(*!
<summary>Runs one typed or borrowed assertion scenario with passive call-local operands.</summary>
<description>
Expected failures are inspected by the independent runner contract suite. Typed entries deliberately receive
literals, properties, arithmetic and method results without intermediate operand variables.
Special floating operands cover exact generic and typed equality and canonical bits at both widths.
Long narrow operands contain ASCII only; their wide counterparts use explicit destination buffer capacities.
</description>
*)
METHOD PROTECTED ExecuteTest
VAR
	value : DINT;
	pointer_ : POINTER TO DINT;
	special : TOF_Core.LREAL_UNION;
	largeUnsigned : ULINT;
	smallerUnsigned : ULINT;
	negativeSigned : LINT;
	zeroUnsigned : ULINT;
	actualReal : REAL;
	expectedReal : REAL;
	realSpecial : TOF_Core.REAL_UNION;
	longAscii : STRING(255);
	longWide : WSTRING(255);
	otherAscii : STRING(255);
	otherWide : WSTRING(255);
	firstLongText : WSTRING(300);
	secondLongText : WSTRING(300);
	subnormalValue : LREAL;
	zeroValue : LREAL;
	subnormalGeneric : TOF_Core.GENERIC_VALUE;
	zeroGeneric : TOF_Core.GENERIC_VALUE;
	subnormalOrder : TOF_Core.COMPARISON_RESULT;
	i : INT;
END_VAR
CASE Scenario OF
	ASSERTION_PROBE_SCENARIO.FLOAT_TOLERANCE:
		Assert.ThatLongReal(actual := LREAL#1.0).ToBe(expected := LREAL#1.0625, tolerance := LREAL#0.125);
		Assert.ThatReal(actual := REAL#1.0).NotToBe(expected := REAL#1.5, tolerance := LREAL#0.125);
		Assert.ThatReal(actual := REAL#1.0).ToBe(expected := REAL#1.0625, tolerance := LREAL#0.125);
		Assert.ThatLongReal(actual := LREAL#1.0).NotToBe(expected := LREAL#1.5, tolerance := LREAL#0.125);
		Assert.ThatReal(actual := REAL#1.0).IsGreaterThanOrEquals(
			expected := REAL#1.0625,
			tolerance := LREAL#0.125
		).IsLessThanOrEquals(expected := REAL#0.9375, tolerance := LREAL#0.125);
		Assert.ThatLongReal(actual := LREAL#1.0).IsGreaterThanOrEquals(
			expected := LREAL#1.0625,
			tolerance := LREAL#0.125
		).IsLessThanOrEquals(expected := LREAL#0.9375, tolerance := LREAL#0.125);
		Assert.ThatLongReal(actual := LREAL#1.0).ToBe(expected := LREAL#1.0, tolerance := TOF_Core.LongReals.ZERO);
		Assert.ThatReal(actual := REAL#1.0).ToBe(
			expected := REAL#1.0625,
			tolerance := LREAL#0.125
		).NotToBe(expected := REAL#1.0625);
		Assert.ThatLongReal(actual := LREAL#1.0).ToBe(
			expected := LREAL#1.0625,
			tolerance := LREAL#0.125
		).NotToBe(expected := LREAL#1.0625);

	ASSERTION_PROBE_SCENARIO.INTEGER_EXACT:
		Assert.ThatULInt(actual := ULINT#9007199254740993).NotToBe(expected := ULINT#9007199254740992);
		Assert.ThatULInt(actual := ULINT#9007199254740993).IsGreaterThan(expected := ULINT#9007199254740992);
		Assert.ThatLInt(actual := LINT#-9223372036854775807).IsLessThan(expected := LINT#-9223372036854775806);
		Assert.ThatULInt(actual := TOF_Core.UnsignedInt64.MAX_VALUE).ToBe(expected := TOF_Core.UnsignedInt64.MAX_VALUE);
		Assert.ThatLInt(actual := TOF_Core.SignedInt64.MIN_VALUE).ToBe(expected := TOF_Core.SignedInt64.MIN_VALUE);
		largeUnsigned := ULINT#9007199254740993;
		smallerUnsigned := ULINT#9007199254740992;
		negativeSigned := LINT#-1;
		zeroUnsigned := TOF_Core.UnsignedInt64.ZERO;
		Assert.That(actual := largeUnsigned).NotToBe(expected := smallerUnsigned);
		Assert.That(actual := largeUnsigned).IsGreaterThan(expected := smallerUnsigned);
		Assert.That(actual := negativeSigned).IsLessThan(expected := zeroUnsigned);

	ASSERTION_PROBE_SCENARIO.TYPED_LITERALS:
		Assert.ThatBool(actual := TRUE).ToBe(expected := TRUE).NotToBe(expected := FALSE).IsTrue();
		Assert.ThatBool(actual := FALSE).IsFalse();
		Assert.ThatSInt(actual := SINT#3)
			.ToBe(expected := SINT#3)
			.NotToBe(expected := SINT#4)
			.IsGreaterThan(expected := SINT#2)
			.IsLessThan(expected := SINT#4)
			.IsGreaterThanOrEquals(expected := SINT#3)
			.IsLessThanOrEquals(expected := SINT#3);
		Assert.ThatInt(actual := INT#3)
			.ToBe(expected := INT#3)
			.NotToBe(expected := INT#4)
			.IsGreaterThan(expected := INT#2)
			.IsLessThan(expected := INT#4)
			.IsGreaterThanOrEquals(expected := INT#3)
			.IsLessThanOrEquals(expected := INT#3);
		Assert.ThatDInt(actual := DINT#3)
			.ToBe(expected := DINT#3)
			.NotToBe(expected := DINT#4)
			.IsGreaterThan(expected := DINT#2)
			.IsLessThan(expected := DINT#4)
			.IsGreaterThanOrEquals(expected := DINT#3)
			.IsLessThanOrEquals(expected := DINT#3);
		Assert.ThatLInt(actual := LINT#3)
			.ToBe(expected := LINT#3)
			.NotToBe(expected := LINT#4)
			.IsGreaterThan(expected := LINT#2)
			.IsLessThan(expected := LINT#4)
			.IsGreaterThanOrEquals(expected := LINT#3)
			.IsLessThanOrEquals(expected := LINT#3);
		Assert.ThatUSInt(actual := USINT#3)
			.ToBe(expected := USINT#3)
			.NotToBe(expected := USINT#4)
			.IsGreaterThan(expected := USINT#2)
			.IsLessThan(expected := USINT#4)
			.IsGreaterThanOrEquals(expected := USINT#3)
			.IsLessThanOrEquals(expected := USINT#3);
		Assert.ThatUInt(actual := UINT#3)
			.ToBe(expected := UINT#3)
			.NotToBe(expected := UINT#4)
			.IsGreaterThan(expected := UINT#2)
			.IsLessThan(expected := UINT#4)
			.IsGreaterThanOrEquals(expected := UINT#3)
			.IsLessThanOrEquals(expected := UINT#3);
		Assert.ThatUDInt(actual := UDINT#3)
			.ToBe(expected := UDINT#3)
			.NotToBe(expected := UDINT#4)
			.IsGreaterThan(expected := UDINT#2)
			.IsLessThan(expected := UDINT#4)
			.IsGreaterThanOrEquals(expected := UDINT#3)
			.IsLessThanOrEquals(expected := UDINT#3);
		Assert.ThatULInt(actual := ULINT#3)
			.ToBe(expected := ULINT#3)
			.NotToBe(expected := ULINT#4)
			.IsGreaterThan(expected := ULINT#2)
			.IsLessThan(expected := ULINT#4)
			.IsGreaterThanOrEquals(expected := ULINT#3)
			.IsLessThanOrEquals(expected := ULINT#3);
		Assert.ThatByte(actual := BYTE#3)
			.ToBe(expected := BYTE#3)
			.NotToBe(expected := BYTE#4)
			.IsGreaterThan(expected := BYTE#2)
			.IsLessThan(expected := BYTE#4)
			.IsGreaterThanOrEquals(expected := BYTE#3)
			.IsLessThanOrEquals(expected := BYTE#3);
		Assert.ThatWord(actual := WORD#3)
			.ToBe(expected := WORD#3)
			.NotToBe(expected := WORD#4)
			.IsGreaterThan(expected := WORD#2)
			.IsLessThan(expected := WORD#4)
			.IsGreaterThanOrEquals(expected := WORD#3)
			.IsLessThanOrEquals(expected := WORD#3);
		Assert.ThatDWord(actual := DWORD#3)
			.ToBe(expected := DWORD#3)
			.NotToBe(expected := DWORD#4)
			.IsGreaterThan(expected := DWORD#2)
			.IsLessThan(expected := DWORD#4)
			.IsGreaterThanOrEquals(expected := DWORD#3)
			.IsLessThanOrEquals(expected := DWORD#3);
		Assert.ThatLWord(actual := LWORD#3)
			.ToBe(expected := LWORD#3)
			.NotToBe(expected := LWORD#4)
			.IsGreaterThan(expected := LWORD#2)
			.IsLessThan(expected := LWORD#4)
			.IsGreaterThanOrEquals(expected := LWORD#3)
			.IsLessThanOrEquals(expected := LWORD#3);
		Assert.ThatReal(actual := REAL#3.0)
			.ToBe(expected := REAL#3.0)
			.NotToBe(expected := REAL#4.0)
			.IsGreaterThan(expected := REAL#2.0)
			.IsLessThan(expected := REAL#4.0)
			.IsGreaterThanOrEquals(expected := REAL#3.0)
			.IsLessThanOrEquals(expected := REAL#3.0);
		Assert.ThatLongReal(actual := LREAL#3.0)
			.ToBe(expected := LREAL#3.0)
			.NotToBe(expected := LREAL#4.0)
			.IsGreaterThan(expected := LREAL#2.0)
			.IsLessThan(expected := LREAL#4.0)
			.IsGreaterThanOrEquals(expected := LREAL#3.0)
			.IsLessThanOrEquals(expected := LREAL#3.0);
		Assert.ThatString(actual := 'b')
			.ToBe(expected := 'b')
			.NotToBe(expected := 'c')
			.IsGreaterThan(expected := 'a')
			.IsLessThan(expected := 'c')
			.IsGreaterThanOrEquals(expected := 'b')
			.IsLessThanOrEquals(expected := 'b');
		Assert.ThatWideString(actual := "b")
			.ToBe(expected := "b")
			.NotToBe(expected := "c")
			.IsGreaterThan(expected := "a")
			.IsLessThan(expected := "c")
			.IsGreaterThanOrEquals(expected := "b")
			.IsLessThanOrEquals(expected := "b");
		Assert.ThatTime(actual := T#3MS)
			.ToBe(expected := T#3MS)
			.NotToBe(expected := T#4MS)
			.IsGreaterThan(expected := T#2MS)
			.IsLessThan(expected := T#4MS)
			.IsGreaterThanOrEquals(expected := T#3MS)
			.IsLessThanOrEquals(expected := T#3MS);
		Assert.ThatLongTime(actual := LTIME#3NS)
			.ToBe(expected := LTIME#3NS)
			.NotToBe(expected := LTIME#4NS)
			.IsGreaterThan(expected := LTIME#2NS)
			.IsLessThan(expected := LTIME#4NS)
			.IsGreaterThanOrEquals(expected := LTIME#3NS)
			.IsLessThanOrEquals(expected := LTIME#3NS);
		Assert.ThatDate(actual := D#2026-11-03)
			.ToBe(expected := D#2026-11-03)
			.NotToBe(expected := D#2026-11-04)
			.IsGreaterThan(expected := D#2026-11-02)
			.IsLessThan(expected := D#2026-11-04)
			.IsGreaterThanOrEquals(expected := D#2026-11-03)
			.IsLessThanOrEquals(expected := D#2026-11-03);
		Assert.ThatLongDate(actual := LDATE#2026-11-03)
			.ToBe(expected := LDATE#2026-11-03)
			.NotToBe(expected := LDATE#2026-11-04)
			.IsGreaterThan(expected := LDATE#2026-11-02)
			.IsLessThan(expected := LDATE#2026-11-04)
			.IsGreaterThanOrEquals(expected := LDATE#2026-11-03)
			.IsLessThanOrEquals(expected := LDATE#2026-11-03);
		Assert.ThatDateTime(actual := DT#2026-11-03-12:00:00)
			.ToBe(expected := DT#2026-11-03-12:00:00)
			.NotToBe(expected := DT#2026-11-03-13:00:00)
			.IsGreaterThan(expected := DT#2026-11-03-11:00:00)
			.IsLessThan(expected := DT#2026-11-03-13:00:00)
			.IsGreaterThanOrEquals(expected := DT#2026-11-03-12:00:00)
			.IsLessThanOrEquals(expected := DT#2026-11-03-12:00:00);
		Assert.ThatLongDateTime(actual := LDT#2026-11-03-12:00:00)
			.ToBe(expected := LDT#2026-11-03-12:00:00)
			.NotToBe(expected := LDT#2026-11-03-13:00:00)
			.IsGreaterThan(expected := LDT#2026-11-03-11:00:00)
			.IsLessThan(expected := LDT#2026-11-03-13:00:00)
			.IsGreaterThanOrEquals(expected := LDT#2026-11-03-12:00:00)
			.IsLessThanOrEquals(expected := LDT#2026-11-03-12:00:00);
		Assert.ThatTimeOfDay(actual := TOD#12:00:00)
			.ToBe(expected := TOD#12:00:00)
			.NotToBe(expected := TOD#13:00:00)
			.IsGreaterThan(expected := TOD#11:00:00)
			.IsLessThan(expected := TOD#13:00:00)
			.IsGreaterThanOrEquals(expected := TOD#12:00:00)
			.IsLessThanOrEquals(expected := TOD#12:00:00);
		Assert.ThatLongTimeOfDay(actual := LTOD#12:00:00)
			.ToBe(expected := LTOD#12:00:00)
			.NotToBe(expected := LTOD#13:00:00)
			.IsGreaterThan(expected := LTOD#11:00:00)
			.IsLessThan(expected := LTOD#13:00:00)
			.IsGreaterThanOrEquals(expected := LTOD#12:00:00)
			.IsLessThanOrEquals(expected := LTOD#12:00:00);
		Assert.ThatDInt(actual := 2 + 3).ToBe(expected := 10 / 2);
		Assert.ThatBool(actual := _Exception.Equals(other := _Exception)).IsTrue();
		Assert.ThatUDInt(actual := CycleCount).IsGreaterThan(expected := TOF_Core.UnsignedInt32.ZERO);
		value := 7;
		Assert.ThatDInt(actual := value).ToBe(expected := replaceValue(value := value));
		Assert.ThatDInt(actual := value).ToBe(expected := 8);

	ASSERTION_PROBE_SCENARIO.MESSAGE_CHAIN:
		Assert.ThatReal(actual := REAL#1.0, message := "Chain diagnostic")
			.IsGreaterThan(expected := REAL#0.5)
			.IsLessThan(expected := REAL#0.5);

	ASSERTION_PROBE_SCENARIO.NEGATIVE_TOLERANCE:
		Assert.ThatReal(actual := REAL#1.0).ToBe(expected := REAL#1.0, tolerance := LREAL#-1.0);

	ASSERTION_PROBE_SCENARIO.NAN_TOLERANCE:
		special.Raw := TOF_Core.LongReals.CANONICAL_NAN_BITS;
		Assert.ThatLongReal(actual := LREAL#1.0).NotToBe(expected := LREAL#2.0, tolerance := special.Value);

	ASSERTION_PROBE_SCENARIO.INFINITE_TOLERANCE:
		Assert.ThatLongReal(actual := LREAL#1.0).IsGreaterThanOrEquals(
			expected := LREAL#0.5,
			tolerance := TOF_Core.LongReals.POSITIVE_INFINITY.Value
		);

	ASSERTION_PROBE_SCENARIO.MESSAGE_RESET:
		Assert.ThatReal(actual := REAL#1.0, message := "Previous diagnostic").ToBe(expected := REAL#1.0);
		Assert.ThatReal(actual := REAL#1.0).ToBe(expected := REAL#2.0);

	ASSERTION_PROBE_SCENARIO.POINTERS_AND_STRINGS:
		Assert.ThatPointer(actual := 0).IsNull().ToBe(expected := 0);
		pointer_ := ADR(value);
		Assert.ThatPointer(actual := pointer_).IsNotNull().ToBe(expected := ADR(value)).NotToBe(expected := 0);
		Assert.That(actual := pointer_).IsNotNull();
		Assert.ThatString(actual := 'abc def').ToContain(substring := 'def');
		Assert.ThatWideString(actual := "abc $042E").ToContain(substring := "$042E");

	ASSERTION_PROBE_SCENARIO.FIRST_FAILURE:
		RecordFailure(message := "First diagnostic");
		Assert.ThatBool(actual := FALSE, message := "Later assertion").IsTrue();

	ASSERTION_PROBE_SCENARIO.SPECIAL_FLOATS:
		checkCanonicalPair(
			realBits := UDINT#16#00000000,
			longRealBits := ULINT#16#8000000000000000,
			expectedBits := ULINT#16#0000000000000000
		);
		checkCanonicalPair(
			realBits := UDINT#16#80000000,
			longRealBits := ULINT#16#0000000000000000,
			expectedBits := ULINT#16#0000000000000000
		);
		checkCanonicalPair(
			realBits := UDINT#16#7F800001,
			longRealBits := ULINT#16#FFF8000000000123,
			expectedBits := ULINT#16#7FF8000000000000
		);
		checkCanonicalPair(
			realBits := UDINT#16#FFC00123,
			longRealBits := ULINT#16#7FF0000000000001,
			expectedBits := ULINT#16#7FF8000000000000
		);
		checkCanonicalPair(
			realBits := UDINT#16#7F800000,
			longRealBits := ULINT#16#7FF0000000000000,
			expectedBits := ULINT#16#7FF0000000000000
		);
		checkCanonicalPair(
			realBits := UDINT#16#FF800000,
			longRealBits := ULINT#16#FFF0000000000000,
			expectedBits := ULINT#16#FFF0000000000000
		);
		checkCanonicalPair(
			realBits := UDINT#16#BFC00000,
			longRealBits := ULINT#16#BFF8000000000000,
			expectedBits := ULINT#16#BFF8000000000000
		);
		checkCanonicalPair(
			realBits := UDINT#16#3F800001,
			longRealBits := ULINT#16#3FF0000020000000,
			expectedBits := ULINT#16#3FF0000020000000
		);

		// The next binary64 value above one rounds to one in binary32.
		actualReal := REAL#1.0;
		special.Raw := ULINT#16#3FF0000000000001;
		Assert.That(actual := actualReal).NotToBe(expected := special.Value);
		Assert.ThatLongReal(actual := LREAL#1.0).NotToBe(expected := special.Value);

		special.Raw := TOF_Core.LongReals.CANONICAL_NAN_BITS;
		Assert.ThatLongReal(actual := special.Value).ToBe(expected := special.Value);
		realSpecial.Raw := UDINT#16#FFC00123;
		expectedReal := realSpecial.Value;
		realSpecial.Raw := UDINT#16#7F800001;
		Assert.That(actual := realSpecial.Value).ToBe(expected := expectedReal);
		Assert.ThatReal(actual := realSpecial.Value)
			.ToBe(expected := expectedReal)
			.IsLessThan(expected := REAL#0.0)
			.IsLessThanOrEquals(expected := realSpecial.Value);
		Assert.ThatReal(actual := REAL#0.0).IsGreaterThan(expected := realSpecial.Value);
		Assert.ThatLongReal(actual := special.Value)
			.IsLessThan(expected := LREAL#0.0)
			.IsGreaterThanOrEquals(expected := special.Value);
		Assert.ThatLongReal(actual := LREAL#0.0).IsGreaterThan(expected := special.Value);

		Assert.ThatLongReal(actual := TOF_Core.LongReals.POSITIVE_INFINITY.Value).ToBe(
			expected := TOF_Core.LongReals.POSITIVE_INFINITY.Value
		);
		Assert.ThatLongReal(actual := TOF_Core.LongReals.POSITIVE_INFINITY.Value).NotToBe(
			expected := TOF_Core.LongReals.NEGATIVE_INFINITY.Value,
			tolerance := LREAL#1.0
		);
		Assert.ThatLongReal(actual := LREAL#-0.0).ToBe(expected := LREAL#0.0);
		Assert.ThatReal(actual := REAL#-0.0).ToBe(expected := REAL#0.0);
		// Binary64 bit 0 encodes the least positive subnormal; default zero tolerance stays canonical.
		special.Raw := ULINT#1;
		Assert.ThatLongReal(actual := special.Value).NotToBe(expected := TOF_Core.LongReals.ZERO);
		subnormalValue := special.Value;
		zeroValue := TOF_Core.LongReals.ZERO;
		subnormalGeneric := TOF_Core.GenericValueFactory.FromAny(
			value := subnormalValue,
			isObject := FALSE,
			memoryManagementBehavior := TOF_Core.GENERIC_MEMORY_MANAGEMENT_BEHAVIOR.STORE_ORIGINAL_REFERENCE_AND_NOT_OWNS_MEMORY
		);
		zeroGeneric := TOF_Core.GenericValueFactory.FromAny(
			value := zeroValue,
			isObject := FALSE,
			memoryManagementBehavior := TOF_Core.GENERIC_MEMORY_MANAGEMENT_BEHAVIOR.STORE_ORIGINAL_REFERENCE_AND_NOT_OWNS_MEMORY
		);
		subnormalOrder := subnormalGeneric.CompareTo(otherValue := zeroGeneric);

		// Core ordering is the oracle for the target's actual handling of subnormal operands.
		IF subnormalOrder <> TOF_Core.COMPARISON_RESULT.FIRST_LESS_THAN_SECOND THEN
			Assert.ThatLongReal(actual := subnormalValue).IsGreaterThanOrEquals(expected := zeroValue);
			Assert.ThatLongReal(actual := zeroValue).IsLessThanOrEquals(expected := subnormalValue);
		END_IF

		IF subnormalOrder <> TOF_Core.COMPARISON_RESULT.FIRST_GREATER_THAN_SECOND THEN
			Assert.ThatLongReal(actual := subnormalValue).IsLessThanOrEquals(expected := zeroValue);
			Assert.ThatLongReal(actual := zeroValue).IsGreaterThanOrEquals(expected := subnormalValue);
		END_IF

	ASSERTION_PROBE_SCENARIO.OPPOSITE_LIMITS:
		Assert.ThatLongReal(actual := TOF_Core.LongReals.MAX_VALUE).NotToBe(
			expected := TOF_Core.LongReals.MIN_VALUE,
			tolerance := TOF_Core.LongReals.MAX_VALUE
		);

	ASSERTION_PROBE_SCENARIO.GENERIC_MESSAGE_CHAIN:
		actualReal := REAL#1.0;
		expectedReal := REAL#0.5;
		Assert.That(actual := actualReal, message := "Generic chain diagnostic")
			.IsGreaterThan(expected := expectedReal)
			.IsLessThan(expected := expectedReal);

	ASSERTION_PROBE_SCENARIO.GENERIC_MESSAGE_RESET:
		actualReal := REAL#1.0;
		expectedReal := REAL#1.0;
		Assert.That(actual := actualReal, message := "Previous generic diagnostic").ToBe(expected := expectedReal);
		expectedReal := REAL#2.0;
		Assert.That(actual := actualReal).ToBe(expected := expectedReal);

	ASSERTION_PROBE_SCENARIO.CONTEXT_TRANSITIONS:
		value := 1;
		actualReal := REAL#1.0;
		Assert.ThatDInt(actual := value, message := "Typed prefix").ToBe(expected := 1);
		Assert.That(actual := value, message := "Generic prefix").NotToBe(expected := actualReal);
		Assert.ThatBool(actual := TRUE).IsTrue();
		Assert.ThatString(actual := 'after generic').ToContain(substring := 'generic');
		Assert.ThatDInt(actual := value).ToBe(expected := 1);

		FOR i := 1 TO 260 DO
			TOF_Core.WideStrings.AppendFit(targetString := firstLongText, sourceString := "x");
		END_FOR

		secondLongText := firstLongText;
		TOF_Core.WideStrings.AppendFit(targetString := firstLongText, sourceString := "A");
		TOF_Core.WideStrings.AppendFit(targetString := secondLongText, sourceString := "B");
		Assert.That(actual := firstLongText).NotToBe(expected := secondLongText);
		Assert.ThatLongReal(actual := LREAL#1.0).ToBe(expected := LREAL#1.0);
		longAscii := TOF_Core.Strings.Concat255(
			'123456789012345678901234567890123456789012345678901234567890123456789012345678901234567890',
			'A'
		);
		otherAscii := TOF_Core.Strings.Concat255(
			'123456789012345678901234567890123456789012345678901234567890123456789012345678901234567890',
			'B'
		);
		Assert.ThatString(actual := longAscii).IsLessThan(expected := otherAscii).NotToBe(expected := otherAscii);
		Assert.ThatString(actual := '').IsLessThan(expected := 'a');
		Assert.ThatString(actual := 'a').IsLessThan(expected := 'aa');
		// Populate wide operands without an intermediate conversion bounded to 80 characters.
		// SA0175: Both sources contain only ASCII; destination capacities include their UTF-16 terminators.
		{analysis -175}
		Tc2_Utilities.STRING_TO_WSTRING2(
			pDstWSTRING := ADR(longWide),
			pSrcSTRING := ADR(longAscii),
			nDstSize := SIZEOF(longWide)
		);
		Tc2_Utilities.STRING_TO_WSTRING2(
			pDstWSTRING := ADR(otherWide),
			pSrcSTRING := ADR(otherAscii),
			nDstSize := SIZEOF(otherWide)
		);
		{analysis +175}
		Assert.ThatWideString(actual := longWide).IsLessThan(expected := otherWide).NotToBe(expected := otherWide);
		Assert.ThatWideString(actual := "$0100").IsGreaterThan(expected := "$00FF");
		Assert.ThatWideString(actual := "").IsLessThan(expected := "a");

	ASSERTION_PROBE_SCENARIO.TYPED_MESSAGE_AFTER_GENERIC:
		value := 1;
		Assert.That(actual := value, message := "Old generic prefix").ToBe(expected := value);
		Assert.ThatByte(actual := BYTE#10, message := "Independent typed").ToBe(expected := BYTE#11);

	ASSERTION_PROBE_SCENARIO.GENERIC_MESSAGE_AFTER_TYPED:
		value := 1;
		largeUnsigned := 2;
		Assert.ThatInt(actual := 1, message := "Old typed prefix").ToBe(expected := 1);
		Assert.That(actual := value, message := "Independent generic").ToBe(expected := largeUnsigned);

	ASSERTION_PROBE_SCENARIO.TYPED_MESSAGE_RESET_AFTER_GENERIC:
		value := 1;
		Assert.ThatDInt(actual := value, message := "Old typed prefix").ToBe(expected := 1);
		Assert.That(actual := value, message := "Old generic prefix").ToBe(expected := value);
		Assert.ThatDInt(actual := value).ToBe(expected := 2);

	ASSERTION_PROBE_SCENARIO.INTEGER_FAILURE:
		Assert.ThatInt(actual := -3).ToBe(expected := -2);

	ASSERTION_PROBE_SCENARIO.BITSTRING_FAILURE:
		Assert.ThatLWord(actual := LWORD#10).ToBe(expected := LWORD#11);

	ASSERTION_PROBE_SCENARIO.POINTER_FAILURE:
		Assert.ThatPointer(actual := ADR(value)).ToBe(expected := TOF_Core.Memory.NULL_ADDRESS);

	ASSERTION_PROBE_SCENARIO.STRING_LONG_FAILURE:
		longAscii := TOF_Core.Strings.Concat255(
			'123456789012345678901234567890123456789012345678901234567890123456789012345678901234567890',
			' ASCII expected suffix'
		);
		Assert.ThatString(actual := 'short').ToBe(expected := longAscii);

	ASSERTION_PROBE_SCENARIO.WIDE_STRING_LONG_FAILURE:
		longWide := TOF_Core.WideStrings.Concat255(
			"123456789012345678901234567890123456789012345678901234567890123456789012345678901234567890",
			" Wide expected suffix"
		);
		Assert.ThatWideString(actual := "short").ToBe(expected := longWide);

	ASSERTION_PROBE_SCENARIO.STRING_CONTAINMENT_FAILURE:
		Assert.ThatString(actual := 'present').ToContain(substring := 'missing');

	ASSERTION_PROBE_SCENARIO.FLOAT_ORDERING_FAILURE:
		realSpecial.Raw := TOF_Core.Reals.CANONICAL_NAN_BITS;
		Assert.ThatReal(actual := realSpecial.Value).IsGreaterThan(expected := REAL#0.0);

	ASSERTION_PROBE_SCENARIO.FLOAT_EQUALITY_FAILURE:
		Assert.ThatReal(actual := REAL#1.0).ToBe(expected := REAL#2.0);

	ASSERTION_PROBE_SCENARIO.TIME_ORDERING_FAILURE:
		Assert.ThatTime(actual := T#1MS).IsGreaterThanOrEquals(expected := T#2MS);
END_CASE
END_METHOD

//! <summary>Borrows the compiler-initialized namespace; callers must not modify the returned reference.</summary>
{attribute 'monitoring' := 'call'}
PROPERTY NamespaceName : REFERENCE TO STRING
GET
NamespaceName REF= _NamespaceName;
END_GET
END_PROPERTY

(*!
<summary>Changes source storage while returning its original value to a typed expected input.</summary>
<description>
Proves that the typed actual operand is a snapshot before evaluation of the next method argument.
</description>
<param name="value">Source variable incremented after its original value is captured.</param>
*)
METHOD PRIVATE replaceValue : DINT
VAR_IN_OUT
	value : DINT;
END_VAR
replaceValue := value;
value := value + 1;
END_METHOD

//! <summary>Reports the complete concrete instance size, excluding separately allocated storage.</summary>
{attribute 'monitoring' := 'call'}
PROPERTY SelfSize : ULINT
GET
SelfSize := XSIZEOF(THIS^);
END_GET
END_PROPERTY

END_FUNCTION_BLOCK

// ---- Tests/Testing/RootTopologyTestRunner.TcPOU
(*
SPDX-License-Identifier: MIT
License: https://opensource.org/license/mit
*)

(*!
<summary>Exercises root topology validation and cyclic execution without repeated scans.</summary>
<description>
Owns persistent root instances and fixed child storage. Use from one task without reentry.
Regression code may deliberately corrupt Children to probe validation; application code must not mutate it.
Children borrows the same array for the instance lifetime. Root parents remain zero.
</description>
*)

{attribute 'no_assign'}
{attribute 'no_explicit_call' := 'do not call this function block directly'}
FUNCTION_BLOCK RootTopologyTestRunner EXTENDS TOF_Testing.TestRunner<2>
VAR_STAT
	//! <summary>Class name shared by instances of this concrete runner.</summary>
	{attribute 'hide'}
	_ClassName : STRING := __POUNAME();
END_VAR
VAR
	{attribute 'hide'}
	{attribute 'init_namespace'}
	_NamespaceName : STRING;
END_VAR
VAR_OUTPUT
	//! <summary>Unregistered owned fixture temporarily placed in a root slot to test active-root rejection.</summary>
	RunningRoot : AssertionIsolationProbe(name := "Running root", parent := 0);
	//! <summary>Owned root element used by this runner.</summary>
	RootTopologyFirst : TestingProbe(name := "Root topology first", parent := 0);
	//! <summary>Owned root element used by this runner.</summary>
	RootTopologyGroup : SingleChildTestGroup(name := "Root topology group", parent := 0);
END_VAR
VAR
	_Children : ARRAY [0.._ChildCount - 1] OF TOF_Testing.ITestElement :=
	[
		RootTopologyFirst,
		RootTopologyGroup
	];
END_VAR

(*!
<summary>Borrows the concrete class name; callers must not modify the returned storage.</summary>
*)
{attribute 'monitoring' := 'call'}
PROPERTY ClassName : REFERENCE TO STRING
GET
ClassName REF= _ClassName;
END_GET
END_PROPERTY

(*!
<summary>Borrows the concrete namespace name for the instance lifetime; callers must not modify it.</summary>
*)
{attribute 'monitoring' := 'call'}
PROPERTY NamespaceName : REFERENCE TO STRING
GET
NamespaceName REF= _NamespaceName;
END_GET
END_PROPERTY

(*!
<summary>Reports the complete concrete instance size.</summary>
*)
{attribute 'monitoring' := 'call'}
PROPERTY SelfSize : ULINT
GET
SelfSize := XSIZEOF(THIS^);
END_GET
END_PROPERTY

(*!
<summary>Borrows the unchanged persistent root array; application code must not modify it.</summary>
*)
{attribute 'monitoring' := 'call'}
PROPERTY Children : REFERENCE TO ARRAY [0.._ChildCount - 1] OF TOF_Testing.ITestElement
GET
Children REF= _Children;
END_GET
END_PROPERTY

END_FUNCTION_BLOCK

// ---- Tests/Testing/MissingChildrenTestGroup.TcPOU
(*
SPDX-License-Identifier: MIT
License: https://opensource.org/license/mit
*)

(*!
<summary>Intentionally omits child-array storage to exercise group validation.</summary>
<description>
Negative fixture: Children intentionally returns an invalid reference without callbacks or exceptions.
Owns no child array or test instances. Use only in the hosting regression task.
</description>
*)

{attribute 'no_assign'}
{attribute 'no_explicit_call' := 'do not call this function block directly'}
FUNCTION_BLOCK MissingChildrenTestGroup EXTENDS TOF_Testing.TestGroup<1>
VAR_STAT
	//! <summary>Class name shared by all instances of this function block.</summary>
	{attribute 'hide'}
	_ClassName : STRING := __POUNAME();
END_VAR
VAR
	{attribute 'hide'}
	{attribute 'init_namespace'}
	_NamespaceName : STRING;
END_VAR

//! <summary>Borrows the concrete class name for the lifetime of this instance; callers must not modify it.</summary>
{attribute 'monitoring' := 'call'}
PROPERTY ClassName : REFERENCE TO STRING
GET
ClassName REF= _ClassName;
END_GET
END_PROPERTY

//! <summary>Borrows the compiler-initialized namespace; callers must not modify the returned reference.</summary>
{attribute 'monitoring' := 'call'}
PROPERTY NamespaceName : REFERENCE TO STRING
GET
NamespaceName REF= _NamespaceName;
END_GET
END_PROPERTY

//! <summary>Reports the complete concrete instance size, excluding separately allocated storage.</summary>
{attribute 'monitoring' := 'call'}
PROPERTY SelfSize : ULINT
GET
SelfSize := XSIZEOF(THIS^);
END_GET
END_PROPERTY

//! <summary>Returns an invalid reference intentionally to exercise missing-storage diagnostics.</summary>
{attribute 'monitoring' := 'call'}
PROPERTY Children : REFERENCE TO ARRAY [0.._ChildCount - 1] OF TOF_Testing.ITestElement
GET
RETURN;
END_GET
END_PROPERTY

END_FUNCTION_BLOCK

// ---- Tests/Testing/MissingChildrenTestRunner.TcPOU
(*
SPDX-License-Identifier: MIT
License: https://opensource.org/license/mit
*)

(*!
<summary>Provides missing root storage for startup and recovery rejection regressions.</summary>
<description>
Deliberately returns an invalid reference to exercise startup and abort-recovery validation.
It owns no roots and provides no backing array. Use only from the hosting regression task.
</description>
*)

{attribute 'no_assign'}
{attribute 'no_explicit_call' := 'do not call this function block directly'}
FUNCTION_BLOCK MissingChildrenTestRunner EXTENDS TOF_Testing.TestRunner<1>
VAR_STAT
	//! <summary>Class name shared by instances of this concrete runner.</summary>
	{attribute 'hide'}
	_ClassName : STRING := __POUNAME();
END_VAR
VAR
	{attribute 'hide'}
	{attribute 'init_namespace'}
	_NamespaceName : STRING;
END_VAR

(*!
<summary>Borrows the concrete class name; callers must not modify the returned storage.</summary>
*)
{attribute 'monitoring' := 'call'}
PROPERTY ClassName : REFERENCE TO STRING
GET
ClassName REF= _ClassName;
END_GET
END_PROPERTY

(*!
<summary>Borrows the concrete namespace name for the instance lifetime; callers must not modify it.</summary>
*)
{attribute 'monitoring' := 'call'}
PROPERTY NamespaceName : REFERENCE TO STRING
GET
NamespaceName REF= _NamespaceName;
END_GET
END_PROPERTY

(*!
<summary>Reports the complete concrete instance size.</summary>
*)
{attribute 'monitoring' := 'call'}
PROPERTY SelfSize : ULINT
GET
SelfSize := XSIZEOF(THIS^);
END_GET
END_PROPERTY

(*!
<summary>Returns an invalid reference for fault injection.</summary>
*)
{attribute 'monitoring' := 'call'}
PROPERTY Children : REFERENCE TO ARRAY [0.._ChildCount - 1] OF TOF_Testing.ITestElement
GET
END_GET
END_PROPERTY

END_FUNCTION_BLOCK

// ---- Tests/Testing/CapturingAdsLogReporter.TcPOU
(*
SPDX-FileCopyrightText: © 2026 Oleksandr Tiutyk <trofimich@gmail.com>
SPDX-License-Identifier: MIT
License: https://opensource.org/license/mit
*)

(*!
<summary>Runs ADS reporter formatting and accounting with a controllable in-memory destination.</summary>
<description>The owning test task selects acceptance before each submission. This fixture performs no ADS I/O.</description>
*)

{attribute 'no_explicit_call' := 'do not call this function block directly'}
FUNCTION_BLOCK CapturingAdsLogReporter EXTENDS TOF_Testing.AdsLogReporter
VAR_STAT
	_CapturingClassName : STRING := __POUNAME();
END_VAR
VAR_INPUT
	//! <summary>Returns FALSE from the destination while this switch is set.</summary>
	RejectWrites : BOOL;
END_VAR
VAR_OUTPUT
	//! <summary>Copies the last accepted message for assertions.</summary>
	AcceptedMessage : TOF_Core.ERROR_MESSAGE;
END_VAR

(*!
<summary>Copies an accepted submission or reports a configured refusal without throwing.</summary>
*)
METHOD PROTECTED TryWriteMessage : BOOL
VAR_INPUT
	category : TOF_Core.LOG_CATEGORY;
END_VAR
VAR_IN_OUT CONSTANT
	message : TOF_Core.ERROR_MESSAGE;
END_VAR
IF RejectWrites THEN
	RETURN;
END_IF

AcceptedMessage := message;
TryWriteMessage := TRUE;
END_METHOD

//! <summary>Provides concrete reporter fixture metadata.</summary>
{attribute 'monitoring' := 'call'}
PROPERTY ClassName : REFERENCE TO STRING
GET
ClassName REF= _CapturingClassName;
END_GET
END_PROPERTY

//! <summary>Reports this concrete fixture size.</summary>
{attribute 'monitoring' := 'call'}
PROPERTY SelfSize : ULINT
GET
SelfSize := XSIZEOF(THIS^);
END_GET
END_PROPERTY

END_FUNCTION_BLOCK

// ---- Tests/Devices/IO/IOModelsTestFixture.TcPOU
(*
SPDX-FileCopyrightText: © 2026 Oleksandr Tiutyk <trofimich@gmail.com>
SPDX-License-Identifier: MIT
License: https://opensource.org/license/mit
*)

(*!
<summary>Holds the existing I/O symbols and runs the model scenarios for the test group.</summary>
<description>
Keep the mapped field names and types at the controller-owned instance path used by the test project.
PDO cases inspect type and byte width through ANY without reading or writing process-image payloads.
Binding cases use fresh local consumers and simulated channels with a live fixture-owned automation parent.
Use from one task. Actual EtherCAT mapping and online change require separate verification.
</description>
*)

{attribute 'no_assign'}
{attribute 'no_explicit_call' := 'do not call this function block directly'}
FUNCTION_BLOCK IOModelsTestFixture IMPLEMENTS IIOModelsTestFixture
VAR_STAT
	{attribute 'hide'}
	_ClassName : STRING := __POUNAME();
END_VAR
VAR CONSTANT
	//! <summary>Bit 6 flags a measurement or hardware error in the simulated channel status word.</summary>
	_ChannelErrorStatus : WORD := WORD#16#0040;
	//! <summary>Initial content outside the simulated fields to expose unintended buffer writes.</summary>
	_UnusedBufferByte : BYTE := BYTE#16#A5;
END_VAR
VAR
	_PulseTrain : TOF_IOModels.EL2521;
	_CounterEncoder : TOF_IOModels.EL5152;
	_LatchedEncoder : TOF_IOModels.EL5151;
	_PowerMeasurement : TOF_IOModels.EL3413_EX;
	_GlobalStatusPowerMeasurement : TOF_IOModels.EL3403;
	_DirectPowerMeasurement : TOF_IOModels.EL3433;
	_Counter : TOF_IOModels.EL1502;
	_Load : TOF_IOModels.EL3356;
	_Pwm : TOF_IOModels.EL2502;
	_Serial : TOF_IOModels.EL6022;
	_DiscreteOutput : TOF_IOModels.EP2624_0002_EX;
	_SixteenChannelInput : TOF_IOModels.EP1809_0021_EX;
	_SixteenChannelOutput : TOF_IOModels.EP2809_0021_EX;
	_MultiRangeInput : TOF_IOModels.EL3078;
	_FieldAnalogInput : TOF_IOModels.EP3174_0002_EX;
	_FieldAnalogOutput : TOF_IOModels.EP4174_0002_EX;
	_FieldSerial : TOF_IOModels.EP6001_0002_EX;

	//! <summary>Live parent borrowed by the simulated analog consumers.</summary>
	_AutomationRoot : MockAutomationController(name := "IOModelsRoot");
END_VAR

(*!
<summary>Runs one IO model scenario and reports to the current case.</summary>
<description>Use from the owning test task. The fixture never retains assertions.</description>
<param name="scenario">Scenario assigned to the caller.</param>
<param name="assertions">Valid assertion context borrowed from the active case.</param>
*)
METHOD ExecuteScenario
VAR_INPUT
	scenario : IO_MODELS_TEST_SCENARIO;
	assertions : REFERENCE TO TOF_Testing.Assertions;
END_VAR
CASE scenario OF
	IO_MODELS_TEST_SCENARIO.PULSE_TRAIN:
		testPulseTrain(assertions := assertions);

	IO_MODELS_TEST_SCENARIO.ENCODER_CHANNELS:
		testEncoderChannels(assertions := assertions);

	IO_MODELS_TEST_SCENARIO.POWER_MEASUREMENT:
		testPowerMeasurement(assertions := assertions);

	IO_MODELS_TEST_SCENARIO.AUXILIARY:
		testAuxiliary(assertions := assertions);

	IO_MODELS_TEST_SCENARIO.COUNTER_AND_LOAD:
		testCounterAndLoad(assertions := assertions);

	IO_MODELS_TEST_SCENARIO.SERIAL_AND_DIAGNOSTICS:
		testSerialAndDiagnostics(assertions := assertions);

	IO_MODELS_TEST_SCENARIO.DISCRETE_CATALOG:
		testDiscreteCatalog(assertions := assertions);

	IO_MODELS_TEST_SCENARIO.ANALOG_REPRESENTATIONS:
		testAnalogRepresentations(assertions := assertions);

	IO_MODELS_TEST_SCENARIO.DINT_BINDING:
		testDintBinding(assertions := assertions);

	IO_MODELS_TEST_SCENARIO.REAL_BINDING:
		testRealBinding(assertions := assertions);
ELSE
	assertions.ThatBool(actual := FALSE, message := "Unknown IO model scenario").IsTrue();
END_CASE
END_METHOD

(*!
<summary>Compares a field descriptor with independent PDO expectations.</summary>
<description>Does not dereference or retain the payload. Pass a model field variable.</description>
<param name="assertions">Valid assertion context of the active case.</param>
<param name="value">Model field whose IEC representation is inspected.</param>
<param name="expectedType">IEC type class required by the selected PDO.</param>
<param name="expectedSize">Required field width in bytes, excluding aggregate padding.</param>
<param name="fieldName">Field identifier used in diagnostic messages.</param>
*)
METHOD PRIVATE checkField
VAR_INPUT
	assertions : REFERENCE TO TOF_Testing.Assertions;
	value : ANY;
	expectedType : __SYSTEM.TYPE_CLASS;
	expectedSize : DINT;
	fieldName : WSTRING(255);
END_VAR
assertions.ThatUDInt(
	actual := TO_UDINT(value.TypeClass),
	message := TOF_Core.WideStrings.Concat255(fieldName, " type")
).ToBe(expected := TO_UDINT(expectedType));
assertions.ThatDInt(
	actual := value.diSize,
	message := TOF_Core.WideStrings.Concat255(fieldName, " byte width")
).ToBe(expected := expectedSize);
END_METHOD

(*!
<summary>Checks the pulse train command and feedback field representations.</summary>
<description>Compares compiler descriptors against independent PDO field expectations.</description>
<param name="assertions">Valid assertion context of the active case.</param>
*)
METHOD PRIVATE testPulseTrain
VAR_INPUT
	assertions : REFERENCE TO TOF_Testing.Assertions;
END_VAR
checkField(
	assertions := assertions,
	value := _PulseTrain.Ch1.Out.Control,
	expectedType := __SYSTEM.TYPE_CLASS.TYPE_WORD,
	expectedSize := 2,
	fieldName := "_PulseTrain.Ch1.Out.Control"
);
checkField(
	assertions := assertions,
	value := _PulseTrain.Ch1.Out.Frequency,
	expectedType := __SYSTEM.TYPE_CLASS.TYPE_UINT,
	expectedSize := 2,
	fieldName := "_PulseTrain.Ch1.Out.Frequency"
);
checkField(
	assertions := assertions,
	value := _PulseTrain.Ch1.Out.TargetCounterValue,
	expectedType := __SYSTEM.TYPE_CLASS.TYPE_UDINT,
	expectedSize := 4,
	fieldName := "_PulseTrain.Ch1.Out.TargetCounterValue"
);
checkField(
	assertions := assertions,
	value := _PulseTrain.Ch1.Out.CounterControl,
	expectedType := __SYSTEM.TYPE_CLASS.TYPE_WORD,
	expectedSize := 2,
	fieldName := "_PulseTrain.Ch1.Out.CounterControl"
);
checkField(
	assertions := assertions,
	value := _PulseTrain.Ch1.Out.SetCounterValue,
	expectedType := __SYSTEM.TYPE_CLASS.TYPE_UDINT,
	expectedSize := 4,
	fieldName := "_PulseTrain.Ch1.Out.SetCounterValue"
);
checkField(
	assertions := assertions,
	value := _PulseTrain.Ch1.In.Status,
	expectedType := __SYSTEM.TYPE_CLASS.TYPE_WORD,
	expectedSize := 2,
	fieldName := "_PulseTrain.Ch1.In.Status"
);
checkField(
	assertions := assertions,
	value := _PulseTrain.Ch1.In.CounterStatus,
	expectedType := __SYSTEM.TYPE_CLASS.TYPE_WORD,
	expectedSize := 2,
	fieldName := "_PulseTrain.Ch1.In.CounterStatus"
);
checkField(
	assertions := assertions,
	value := _PulseTrain.Ch1.In.CounterValue,
	expectedType := __SYSTEM.TYPE_CLASS.TYPE_UDINT,
	expectedSize := 4,
	fieldName := "_PulseTrain.Ch1.In.CounterValue"
);
END_METHOD

(*!
<summary>Checks counter and latched encoder command and feedback field representations.</summary>
<description>Compares compiler descriptors against independent PDO field expectations.</description>
<param name="assertions">Valid assertion context of the active case.</param>
*)
METHOD PRIVATE testEncoderChannels
VAR_INPUT
	assertions : REFERENCE TO TOF_Testing.Assertions;
END_VAR
checkField(
	assertions := assertions,
	value := _CounterEncoder.Ch1.In.Status,
	expectedType := __SYSTEM.TYPE_CLASS.TYPE_WORD,
	expectedSize := 2,
	fieldName := "_CounterEncoder.Ch1.In.Status"
);
checkField(
	assertions := assertions,
	value := _CounterEncoder.Ch1.In.Value,
	expectedType := __SYSTEM.TYPE_CLASS.TYPE_UDINT,
	expectedSize := 4,
	fieldName := "_CounterEncoder.Ch1.In.Value"
);
checkField(
	assertions := assertions,
	value := _CounterEncoder.Ch2.In.Value,
	expectedType := __SYSTEM.TYPE_CLASS.TYPE_UDINT,
	expectedSize := 4,
	fieldName := "_CounterEncoder.Ch2.In.Value"
);
checkField(
	assertions := assertions,
	value := _CounterEncoder.Ch1.Out.SetValue,
	expectedType := __SYSTEM.TYPE_CLASS.TYPE_UDINT,
	expectedSize := 4,
	fieldName := "_CounterEncoder.Ch1.Out.SetValue"
);
checkField(
	assertions := assertions,
	value := _LatchedEncoder.Ch1.In.Latch,
	expectedType := __SYSTEM.TYPE_CLASS.TYPE_UDINT,
	expectedSize := 4,
	fieldName := "_LatchedEncoder.Ch1.In.Latch"
);
checkField(
	assertions := assertions,
	value := _LatchedEncoder.Ch1.Out.Control,
	expectedType := __SYSTEM.TYPE_CLASS.TYPE_WORD,
	expectedSize := 2,
	fieldName := "_LatchedEncoder.Ch1.Out.Control"
);
END_METHOD

(*!
<summary>Checks selected channel fields in the three power measurement models.</summary>
<description>Compares compiler descriptors against independent PDO field expectations.</description>
<param name="assertions">Valid assertion context of the active case.</param>
*)
METHOD PRIVATE testPowerMeasurement
VAR_INPUT
	assertions : REFERENCE TO TOF_Testing.Assertions;
END_VAR
checkField(
	assertions := assertions,
	value := _PowerMeasurement.L1.In.Status,
	expectedType := __SYSTEM.TYPE_CLASS.TYPE_WORD,
	expectedSize := 2,
	fieldName := "_PowerMeasurement.L1.In.Status"
);
checkField(
	assertions := assertions,
	value := _PowerMeasurement.L1.In.Current,
	expectedType := __SYSTEM.TYPE_CLASS.TYPE_DINT,
	expectedSize := 4,
	fieldName := "_PowerMeasurement.L1.In.Current"
);
checkField(
	assertions := assertions,
	value := _PowerMeasurement.L1.In.Voltage,
	expectedType := __SYSTEM.TYPE_CLASS.TYPE_DINT,
	expectedSize := 4,
	fieldName := "_PowerMeasurement.L1.In.Voltage"
);
checkField(
	assertions := assertions,
	value := _PowerMeasurement.L1.In.ActivePower,
	expectedType := __SYSTEM.TYPE_CLASS.TYPE_DINT,
	expectedSize := 4,
	fieldName := "_PowerMeasurement.L1.In.ActivePower"
);
checkField(
	assertions := assertions,
	value := _PowerMeasurement.L1.In.Index,
	expectedType := __SYSTEM.TYPE_CLASS.TYPE_USINT,
	expectedSize := 1,
	fieldName := "_PowerMeasurement.L1.In.Index"
);
checkField(
	assertions := assertions,
	value := _PowerMeasurement.L1.In.VariantValue,
	expectedType := __SYSTEM.TYPE_CLASS.TYPE_DINT,
	expectedSize := 4,
	fieldName := "_PowerMeasurement.L1.In.VariantValue"
);
checkField(
	assertions := assertions,
	value := _GlobalStatusPowerMeasurement.L1.In.Status,
	expectedType := __SYSTEM.TYPE_CLASS.TYPE_WORD,
	expectedSize := 2,
	fieldName := "_GlobalStatusPowerMeasurement.L1.In.Status"
);
checkField(
	assertions := assertions,
	value := _GlobalStatusPowerMeasurement.L1.In.Current,
	expectedType := __SYSTEM.TYPE_CLASS.TYPE_DINT,
	expectedSize := 4,
	fieldName := "_GlobalStatusPowerMeasurement.L1.In.Current"
);
checkField(
	assertions := assertions,
	value := _GlobalStatusPowerMeasurement.L1.In.Voltage,
	expectedType := __SYSTEM.TYPE_CLASS.TYPE_DINT,
	expectedSize := 4,
	fieldName := "_GlobalStatusPowerMeasurement.L1.In.Voltage"
);
checkField(
	assertions := assertions,
	value := _GlobalStatusPowerMeasurement.Status,
	expectedType := __SYSTEM.TYPE_CLASS.TYPE_WORD,
	expectedSize := 2,
	fieldName := "_GlobalStatusPowerMeasurement.Status"
);
END_METHOD

(*!
<summary>Checks auxiliary power measurement and PWM field representations.</summary>
<description>Compares compiler descriptors against independent PDO field expectations.</description>
<param name="assertions">Valid assertion context of the active case.</param>
*)
METHOD PRIVATE testAuxiliary
VAR_INPUT
	assertions : REFERENCE TO TOF_Testing.Assertions;
END_VAR
checkField(
	assertions := assertions,
	value := _PowerMeasurement.Auxiliary.In.Status,
	expectedType := __SYSTEM.TYPE_CLASS.TYPE_WORD,
	expectedSize := 2,
	fieldName := "_PowerMeasurement.Auxiliary.In.Status"
);
checkField(
	assertions := assertions,
	value := _PowerMeasurement.Auxiliary.In.Index,
	expectedType := __SYSTEM.TYPE_CLASS.TYPE_USINT,
	expectedSize := 1,
	fieldName := "_PowerMeasurement.Auxiliary.In.Index"
);
checkField(
	assertions := assertions,
	value := _PowerMeasurement.Auxiliary.In.Channel,
	expectedType := __SYSTEM.TYPE_CLASS.TYPE_USINT,
	expectedSize := 1,
	fieldName := "_PowerMeasurement.Auxiliary.In.Channel"
);
checkField(
	assertions := assertions,
	value := _PowerMeasurement.Auxiliary.In.Value,
	expectedType := __SYSTEM.TYPE_CLASS.TYPE_DINT,
	expectedSize := 4,
	fieldName := "_PowerMeasurement.Auxiliary.In.Value"
);
checkField(
	assertions := assertions,
	value := _PowerMeasurement.Auxiliary.Out.Index,
	expectedType := __SYSTEM.TYPE_CLASS.TYPE_USINT,
	expectedSize := 1,
	fieldName := "_PowerMeasurement.Auxiliary.Out.Index"
);
checkField(
	assertions := assertions,
	value := _PowerMeasurement.Auxiliary.Out.Channel,
	expectedType := __SYSTEM.TYPE_CLASS.TYPE_USINT,
	expectedSize := 1,
	fieldName := "_PowerMeasurement.Auxiliary.Out.Channel"
);
checkField(
	assertions := assertions,
	value := _DirectPowerMeasurement.Auxiliary.In.Value,
	expectedType := __SYSTEM.TYPE_CLASS.TYPE_DINT,
	expectedSize := 4,
	fieldName := "_DirectPowerMeasurement.Auxiliary.In.Value"
);
END_METHOD

(*!
<summary>Checks counter and load cell field representations.</summary>
<description>Compares compiler descriptors against independent PDO field expectations.</description>
<param name="assertions">Valid assertion context of the active case.</param>
*)
METHOD PRIVATE testCounterAndLoad
VAR_INPUT
	assertions : REFERENCE TO TOF_Testing.Assertions;
END_VAR
checkField(
	assertions := assertions,
	value := _Counter.Ch1.In.Status,
	expectedType := __SYSTEM.TYPE_CLASS.TYPE_WORD,
	expectedSize := 2,
	fieldName := "_Counter.Ch1.In.Status"
);
checkField(
	assertions := assertions,
	value := _Counter.Ch1.In.CounterValue,
	expectedType := __SYSTEM.TYPE_CLASS.TYPE_UDINT,
	expectedSize := 4,
	fieldName := "_Counter.Ch1.In.CounterValue"
);
checkField(
	assertions := assertions,
	value := _Counter.Ch1.Out.Control,
	expectedType := __SYSTEM.TYPE_CLASS.TYPE_WORD,
	expectedSize := 2,
	fieldName := "_Counter.Ch1.Out.Control"
);
checkField(
	assertions := assertions,
	value := _Counter.Ch1.Out.SetCounterValue,
	expectedType := __SYSTEM.TYPE_CLASS.TYPE_UDINT,
	expectedSize := 4,
	fieldName := "_Counter.Ch1.Out.SetCounterValue"
);
checkField(
	assertions := assertions,
	value := _Load.Ch1.In.Status,
	expectedType := __SYSTEM.TYPE_CLASS.TYPE_WORD,
	expectedSize := 2,
	fieldName := "_Load.Ch1.In.Status"
);
checkField(
	assertions := assertions,
	value := _Load.Ch1.In.Value,
	expectedType := __SYSTEM.TYPE_CLASS.TYPE_DINT,
	expectedSize := 4,
	fieldName := "_Load.Ch1.In.Value"
);
checkField(
	assertions := assertions,
	value := _Load.Ch1.Out.Control,
	expectedType := __SYSTEM.TYPE_CLASS.TYPE_WORD,
	expectedSize := 2,
	fieldName := "_Load.Ch1.Out.Control"
);
checkField(
	assertions := assertions,
	value := _Pwm.Ch1.DutyCycle,
	expectedType := __SYSTEM.TYPE_CLASS.TYPE_INT,
	expectedSize := 2,
	fieldName := "_Pwm.Ch1.DutyCycle"
);
END_METHOD

(*!
<summary>Checks serial payload widths and diagnostics on selected models.</summary>
<description>Compares compiler descriptors against independent PDO field expectations.</description>
<param name="assertions">Valid assertion context of the active case.</param>
*)
METHOD PRIVATE testSerialAndDiagnostics
VAR_INPUT
	assertions : REFERENCE TO TOF_Testing.Assertions;
END_VAR
checkField(
	assertions := assertions,
	value := _Serial.Ch1.InData.Status,
	expectedType := __SYSTEM.TYPE_CLASS.TYPE_WORD,
	expectedSize := 2,
	fieldName := "_Serial.Ch1.InData.Status"
);
checkField(
	assertions := assertions,
	value := _Serial.Ch1.OutData.Control,
	expectedType := __SYSTEM.TYPE_CLASS.TYPE_WORD,
	expectedSize := 2,
	fieldName := "_Serial.Ch1.OutData.Control"
);
checkField(
	assertions := assertions,
	value := _PowerMeasurement.WcState,
	expectedType := __SYSTEM.TYPE_CLASS.TYPE_BOOL,
	expectedSize := 1,
	fieldName := "_PowerMeasurement.WcState"
);
checkField(
	assertions := assertions,
	value := _PowerMeasurement.InputToggle,
	expectedType := __SYSTEM.TYPE_CLASS.TYPE_BOOL,
	expectedSize := 1,
	fieldName := "_PowerMeasurement.InputToggle"
);
checkField(
	assertions := assertions,
	value := _PowerMeasurement.State,
	expectedType := __SYSTEM.TYPE_CLASS.TYPE_UINT,
	expectedSize := 2,
	fieldName := "_PowerMeasurement.State"
);
checkField(
	assertions := assertions,
	value := _DiscreteOutput.WcState,
	expectedType := __SYSTEM.TYPE_CLASS.TYPE_BOOL,
	expectedSize := 1,
	fieldName := "_DiscreteOutput.WcState"
);
checkField(
	assertions := assertions,
	value := _DiscreteOutput.State,
	expectedType := __SYSTEM.TYPE_CLASS.TYPE_UINT,
	expectedSize := 2,
	fieldName := "_DiscreteOutput.State"
);
assertions.ThatUDInt(
	actual := SIZEOF(_Serial.Ch1.InData.Data),
	message := "Serial receive payload is 22 bytes"
).ToBe(expected := 22);
assertions.ThatUDInt(
	actual := SIZEOF(_Serial.Ch1.OutData.Data),
	message := "Serial transmit payload is 22 bytes"
).ToBe(expected := 22);
assertions.ThatUDInt(
	actual := SIZEOF(_PowerMeasurement.AdsAddr),
	message := "ADS address is NetId plus port"
).ToBe(expected := 8);
END_METHOD

(*!
<summary>Checks the corrected 16-channel EP product types and their boundary endpoints.</summary>
<description>Compares compiler descriptors against independent PDO field expectations.</description>
<param name="assertions">Valid assertion context of the active case.</param>
*)
METHOD PRIVATE testDiscreteCatalog
VAR_INPUT
	assertions : REFERENCE TO TOF_Testing.Assertions;
END_VAR
checkField(
	assertions := assertions,
	value := _SixteenChannelInput.Ch01,
	expectedType := __SYSTEM.TYPE_CLASS.TYPE_BOOL,
	expectedSize := 1,
	fieldName := "_SixteenChannelInput.Ch01"
);
checkField(
	assertions := assertions,
	value := _SixteenChannelInput.Ch16,
	expectedType := __SYSTEM.TYPE_CLASS.TYPE_BOOL,
	expectedSize := 1,
	fieldName := "_SixteenChannelInput.Ch16"
);
checkField(
	assertions := assertions,
	value := _SixteenChannelInput.WcState,
	expectedType := __SYSTEM.TYPE_CLASS.TYPE_BOOL,
	expectedSize := 1,
	fieldName := "_SixteenChannelInput.WcState"
);
checkField(
	assertions := assertions,
	value := _SixteenChannelInput.InputToggle,
	expectedType := __SYSTEM.TYPE_CLASS.TYPE_BOOL,
	expectedSize := 1,
	fieldName := "_SixteenChannelInput.InputToggle"
);
checkField(
	assertions := assertions,
	value := _SixteenChannelInput.State,
	expectedType := __SYSTEM.TYPE_CLASS.TYPE_UINT,
	expectedSize := 2,
	fieldName := "_SixteenChannelInput.State"
);
checkField(
	assertions := assertions,
	value := _SixteenChannelOutput.Ch01,
	expectedType := __SYSTEM.TYPE_CLASS.TYPE_BOOL,
	expectedSize := 1,
	fieldName := "_SixteenChannelOutput.Ch01"
);
checkField(
	assertions := assertions,
	value := _SixteenChannelOutput.Ch16,
	expectedType := __SYSTEM.TYPE_CLASS.TYPE_BOOL,
	expectedSize := 1,
	fieldName := "_SixteenChannelOutput.Ch16"
);
checkField(
	assertions := assertions,
	value := _SixteenChannelOutput.WcState,
	expectedType := __SYSTEM.TYPE_CLASS.TYPE_BOOL,
	expectedSize := 1,
	fieldName := "_SixteenChannelOutput.WcState"
);
checkField(
	assertions := assertions,
	value := _SixteenChannelOutput.State,
	expectedType := __SYSTEM.TYPE_CLASS.TYPE_UINT,
	expectedSize := 2,
	fieldName := "_SixteenChannelOutput.State"
);
checkField(
	assertions := assertions,
	value := _DiscreteOutput.Ch1,
	expectedType := __SYSTEM.TYPE_CLASS.TYPE_BOOL,
	expectedSize := 1,
	fieldName := "_DiscreteOutput.Ch1"
);
checkField(
	assertions := assertions,
	value := _DiscreteOutput.Ch4,
	expectedType := __SYSTEM.TYPE_CLASS.TYPE_BOOL,
	expectedSize := 1,
	fieldName := "_DiscreteOutput.Ch4"
);
END_METHOD

(*!
<summary>Checks EL3078 Real32 and the analog and serial EP endpoints.</summary>
<description>Compares compiler descriptors against independent PDO field expectations.</description>
<param name="assertions">Valid assertion context of the active case.</param>
*)
METHOD PRIVATE testAnalogRepresentations
VAR_INPUT
	assertions : REFERENCE TO TOF_Testing.Assertions;
END_VAR
checkField(
	assertions := assertions,
	value := _MultiRangeInput.Ch1.Status,
	expectedType := __SYSTEM.TYPE_CLASS.TYPE_WORD,
	expectedSize := 2,
	fieldName := "_MultiRangeInput.Ch1.Status"
);
checkField(
	assertions := assertions,
	value := _MultiRangeInput.Ch1.Value,
	expectedType := __SYSTEM.TYPE_CLASS.TYPE_REAL,
	expectedSize := 4,
	fieldName := "_MultiRangeInput.Ch1.Value"
);
checkField(
	assertions := assertions,
	value := _MultiRangeInput.Ch8.Status,
	expectedType := __SYSTEM.TYPE_CLASS.TYPE_WORD,
	expectedSize := 2,
	fieldName := "_MultiRangeInput.Ch8.Status"
);
checkField(
	assertions := assertions,
	value := _MultiRangeInput.Ch8.Value,
	expectedType := __SYSTEM.TYPE_CLASS.TYPE_REAL,
	expectedSize := 4,
	fieldName := "_MultiRangeInput.Ch8.Value"
);
checkField(
	assertions := assertions,
	value := _FieldAnalogInput.Ch4.Status,
	expectedType := __SYSTEM.TYPE_CLASS.TYPE_WORD,
	expectedSize := 2,
	fieldName := "_FieldAnalogInput.Ch4.Status"
);
checkField(
	assertions := assertions,
	value := _FieldAnalogInput.Ch4.Value,
	expectedType := __SYSTEM.TYPE_CLASS.TYPE_INT,
	expectedSize := 2,
	fieldName := "_FieldAnalogInput.Ch4.Value"
);
checkField(
	assertions := assertions,
	value := _FieldAnalogOutput.Ch4,
	expectedType := __SYSTEM.TYPE_CLASS.TYPE_INT,
	expectedSize := 2,
	fieldName := "_FieldAnalogOutput.Ch4"
);
checkField(
	assertions := assertions,
	value := _FieldSerial.Ch1.InData.Status,
	expectedType := __SYSTEM.TYPE_CLASS.TYPE_WORD,
	expectedSize := 2,
	fieldName := "_FieldSerial.Ch1.InData.Status"
);
checkField(
	assertions := assertions,
	value := _FieldSerial.Ch1.OutData.Control,
	expectedType := __SYSTEM.TYPE_CLASS.TYPE_WORD,
	expectedSize := 2,
	fieldName := "_FieldSerial.Ch1.OutData.Control"
);

assertions.ThatUDInt(
	actual := SIZEOF(_FieldAnalogInput.AdsAddr),
	message := "_FieldAnalogInput retains the supported CoE ADS endpoint"
).ToBe(expected := 8);
assertions.ThatUDInt(
	actual := SIZEOF(_FieldAnalogOutput.AdsAddr),
	message := "_FieldAnalogOutput retains the supported CoE ADS endpoint"
).ToBe(expected := 8);
assertions.ThatUDInt(
	actual := SIZEOF(_FieldSerial.AdsAddr),
	message := "_FieldSerial retains the supported CoE ADS endpoint"
).ToBe(expected := 8);
END_METHOD

(*!
<summary>Checks signed DINT input binding, recovery, unbinding and source preservation.</summary>
<description>Builds a fresh simulated channel in ordinary storage. Offsets describe the PLC layout.</description>
<param name="assertions">Valid assertion context of the active case.</param>
*)
METHOD PRIVATE testDintBinding
VAR_INPUT
	assertions : REFERENCE TO TOF_Testing.Assertions;
END_VAR
VAR
	converter : TOF_Devices_IO.DirectAnalogValueConverter;
	analogInput : TOF_Devices_IO.AnalogInput(
		name := "DintModelInput",
		parent := _AutomationRoot,
		converter := converter
	);
	channelStorage : ARRAY [0..31] OF BYTE;
	unboundChannel : REFERENCE TO TOF_IOModels.ANALOG_INPUT_DINT_CHANNEL;
	channel : POINTER TO TOF_IOModels.ANALOG_INPUT_DINT_CHANNEL;
	rawValue : DINT;
	rawStatus : WORD;
	valueOffset : UDINT;
	statusOffset : UDINT;
	originalBytes : ARRAY [0..31] OF BYTE;
	i : DINT;
END_VAR
channel := ADR(channelStorage);

IF SIZEOF(channel^) > SIZEOF(channelStorage) THEN
	assertions.ThatBool(
		actual := FALSE,
		message := "Simulated channel storage is too small"
	).IsTrue();

	RETURN;
END_IF

valueOffset := TO_UDINT(ADR(channel^.Value) - ADR(channel^));
statusOffset := TO_UDINT(ADR(channel^.Status) - ADR(channel^));

FOR i := LOWER_BOUND(channelStorage, 1) TO UPPER_BOUND(channelStorage, 1) DO
	channelStorage[i] := _UnusedBufferByte;
END_FOR

rawValue := DINT#-123456789;
rawStatus := WORD#0;
Tc2_System.MEMCPY(
	destAddr := ADR(channelStorage[valueOffset]),
	srcAddr := ADR(rawValue),
	n := SIZEOF(rawValue)
);
Tc2_System.MEMCPY(
	destAddr := ADR(channelStorage[statusOffset]),
	srcAddr := ADR(rawStatus),
	n := SIZEOF(rawStatus)
);

FOR i := LOWER_BOUND(channelStorage, 1) TO UPPER_BOUND(channelStorage, 1) DO
	originalBytes[i] := channelStorage[i];
END_FOR

IF NOT analogInput.Initialize() THEN
	assertions.ThatBool(actual := FALSE, message := "The analog input must initialize").IsTrue();

	RETURN;
END_IF

analogInput.BindToInt32IO(rawValues := channel^);
analogInput.ProcessInput();
assertions.ThatBool(
	actual := analogInput.BoundToIO,
	message := "Valid channel must bind"
).IsTrue();
assertions.ThatLongReal(
	actual := analogInput.Value,
	message := "The signed DINT value must survive binding"
).ToBe(expected := LREAL#-123456789.0);

FOR i := LOWER_BOUND(channelStorage, 1) TO UPPER_BOUND(channelStorage, 1) DO
	assertions.ThatByte(
		actual := channelStorage[i],
		message := TOF_Core.WideStrings.Concat255("Binding and processing changed byte ", TO_WSTRING(i))
	).ToBe(expected := originalBytes[i]);
END_FOR

rawStatus := _ChannelErrorStatus;
Tc2_System.MEMCPY(
	destAddr := ADR(channelStorage[statusOffset]),
	srcAddr := ADR(rawStatus),
	n := SIZEOF(rawStatus)
);
analogInput.ProcessInput();
assertions.ThatBool(
	actual := analogInput.HasError,
	message := "Live channel error must be reported"
).IsTrue();
assertions.ThatBool(
	actual := analogInput.Status.Error,
	message := "Live channel must expose the sampled error bit"
).IsTrue();
analogInput.BindToInt32IO(rawValues := unboundChannel);
analogInput.ProcessInput();
assertions.ThatBool(
	actual := analogInput.BoundToIO,
	message := "Invalid reference must unbind value"
).IsFalse();
assertions.ThatBool(
	actual := analogInput.Status.Error,
	message := "Invalid reference must unbind status"
).IsFalse();

rawValue := DINT#7654321;
rawStatus := WORD#0;
Tc2_System.MEMCPY(
	destAddr := ADR(channelStorage[valueOffset]),
	srcAddr := ADR(rawValue),
	n := SIZEOF(rawValue)
);
Tc2_System.MEMCPY(
	destAddr := ADR(channelStorage[statusOffset]),
	srcAddr := ADR(rawStatus),
	n := SIZEOF(rawStatus)
);

FOR i := LOWER_BOUND(channelStorage, 1) TO UPPER_BOUND(channelStorage, 1) DO
	originalBytes[i] := channelStorage[i];
END_FOR

analogInput.BindToInt32IO(rawValues := channel^);
analogInput.ProcessInput();
assertions.ThatBool(
	actual := analogInput.BoundToIO,
	message := "Recovered channel must bind again"
).IsTrue();
assertions.ThatLongReal(
	actual := analogInput.Value,
	message := "Rebinding must read the updated source"
).ToBe(expected := LREAL#7654321.0);
assertions.ThatBool(
	actual := analogInput.HasError,
	message := "Rebinding to recovered status must clear error"
).IsFalse();
analogInput.BindToInt32IO(rawValues := unboundChannel);

FOR i := LOWER_BOUND(channelStorage, 1) TO UPPER_BOUND(channelStorage, 1) DO
	assertions.ThatByte(
		actual := channelStorage[i],
		message := TOF_Core.WideStrings.Concat255(
			"Rebinding, processing or unbinding changed byte ",
			TO_WSTRING(i)
		)
	).ToBe(expected := originalBytes[i]);
END_FOR
END_METHOD

(*!
<summary>Checks fractional REAL input binding, recovery, unbinding and source preservation.</summary>
<description>Builds a fresh simulated channel in ordinary storage. Offsets describe the PLC layout.</description>
<param name="assertions">Valid assertion context of the active case.</param>
*)
METHOD PRIVATE testRealBinding
VAR_INPUT
	assertions : REFERENCE TO TOF_Testing.Assertions;
END_VAR
VAR
	converter : TOF_Devices_IO.DirectAnalogValueConverter;
	analogInput : TOF_Devices_IO.AnalogInput(
		name := "RealModelInput",
		parent := _AutomationRoot,
		converter := converter
	);
	channelStorage : ARRAY [0..31] OF BYTE;
	unboundChannel : REFERENCE TO TOF_IOModels.ANALOG_INPUT_REAL_CHANNEL;
	channel : POINTER TO TOF_IOModels.ANALOG_INPUT_REAL_CHANNEL;
	rawValue : REAL;
	rawStatus : WORD;
	valueOffset : UDINT;
	statusOffset : UDINT;
	originalBytes : ARRAY [0..31] OF BYTE;
	i : DINT;
END_VAR
channel := ADR(channelStorage);

IF SIZEOF(channel^) > SIZEOF(channelStorage) THEN
	assertions.ThatBool(
		actual := FALSE,
		message := "Simulated channel storage is too small"
	).IsTrue();

	RETURN;
END_IF

valueOffset := TO_UDINT(ADR(channel^.Value) - ADR(channel^));
statusOffset := TO_UDINT(ADR(channel^.Status) - ADR(channel^));

FOR i := LOWER_BOUND(channelStorage, 1) TO UPPER_BOUND(channelStorage, 1) DO
	channelStorage[i] := _UnusedBufferByte;
END_FOR

rawValue := REAL#-12.75;
rawStatus := WORD#0;
Tc2_System.MEMCPY(
	destAddr := ADR(channelStorage[valueOffset]),
	srcAddr := ADR(rawValue),
	n := SIZEOF(rawValue)
);
Tc2_System.MEMCPY(
	destAddr := ADR(channelStorage[statusOffset]),
	srcAddr := ADR(rawStatus),
	n := SIZEOF(rawStatus)
);

FOR i := LOWER_BOUND(channelStorage, 1) TO UPPER_BOUND(channelStorage, 1) DO
	originalBytes[i] := channelStorage[i];
END_FOR

IF NOT analogInput.Initialize() THEN
	assertions.ThatBool(actual := FALSE, message := "The analog input must initialize").IsTrue();

	RETURN;
END_IF

analogInput.BindToReal32IO(rawValues := channel^);
analogInput.ProcessInput();
assertions.ThatBool(
	actual := analogInput.BoundToIO,
	message := "Valid channel must bind"
).IsTrue();
assertions.ThatLongReal(
	actual := analogInput.Value,
	message := "The fractional REAL value must survive binding"
).ToBe(expected := LREAL#-12.75);

FOR i := LOWER_BOUND(channelStorage, 1) TO UPPER_BOUND(channelStorage, 1) DO
	assertions.ThatByte(
		actual := channelStorage[i],
		message := TOF_Core.WideStrings.Concat255("Binding and processing changed byte ", TO_WSTRING(i))
	).ToBe(expected := originalBytes[i]);
END_FOR

rawStatus := _ChannelErrorStatus;
Tc2_System.MEMCPY(
	destAddr := ADR(channelStorage[statusOffset]),
	srcAddr := ADR(rawStatus),
	n := SIZEOF(rawStatus)
);
analogInput.ProcessInput();
assertions.ThatBool(
	actual := analogInput.HasError,
	message := "Live channel error must be reported"
).IsTrue();
assertions.ThatBool(
	actual := analogInput.Status.Error,
	message := "Live channel must expose the sampled error bit"
).IsTrue();
analogInput.BindToReal32IO(rawValues := unboundChannel);
analogInput.ProcessInput();
assertions.ThatBool(
	actual := analogInput.BoundToIO,
	message := "Invalid reference must unbind value"
).IsFalse();
assertions.ThatBool(
	actual := analogInput.Status.Error,
	message := "Invalid reference must unbind status"
).IsFalse();

rawValue := REAL#23.5;
rawStatus := WORD#0;
Tc2_System.MEMCPY(
	destAddr := ADR(channelStorage[valueOffset]),
	srcAddr := ADR(rawValue),
	n := SIZEOF(rawValue)
);
Tc2_System.MEMCPY(
	destAddr := ADR(channelStorage[statusOffset]),
	srcAddr := ADR(rawStatus),
	n := SIZEOF(rawStatus)
);

FOR i := LOWER_BOUND(channelStorage, 1) TO UPPER_BOUND(channelStorage, 1) DO
	originalBytes[i] := channelStorage[i];
END_FOR

analogInput.BindToReal32IO(rawValues := channel^);
analogInput.ProcessInput();
assertions.ThatBool(
	actual := analogInput.BoundToIO,
	message := "Recovered channel must bind again"
).IsTrue();
assertions.ThatLongReal(
	actual := analogInput.Value,
	message := "Rebinding must read the updated source"
).ToBe(expected := LREAL#23.5);
assertions.ThatBool(
	actual := analogInput.HasError,
	message := "Rebinding to recovered status must clear error"
).IsFalse();
analogInput.BindToReal32IO(rawValues := unboundChannel);

FOR i := LOWER_BOUND(channelStorage, 1) TO UPPER_BOUND(channelStorage, 1) DO
	assertions.ThatByte(
		actual := channelStorage[i],
		message := TOF_Core.WideStrings.Concat255(
			"Rebinding, processing or unbinding changed byte ",
			TO_WSTRING(i)
		)
	).ToBe(expected := originalBytes[i]);
END_FOR
END_METHOD

END_FUNCTION_BLOCK

// ---- Tests/Automation/MockAutomationController.TcPOU
(*
SPDX-FileCopyrightText: © 2026 Oleksandr Tiutyk <trofimich@gmail.com>
SPDX-License-Identifier: MIT
License: https://opensource.org/license/mit
*)

(*!
<summary>Mock root controller for automation component lifecycle and hierarchy tests.</summary>
*)

FUNCTION_BLOCK MockAutomationController EXTENDS TOF_Automation.AutomationController<0>
VAR_STAT
	{attribute 'hide'}
	_ClassName : STRING := __POUNAME();
END_VAR

PROPERTY Children : REFERENCE TO ARRAY [0.._ChildCount - 1] OF TOF_Automation.IChildAutomationComponent
GET
Children REF= 0;
END_GET
END_PROPERTY

{attribute 'monitoring' := 'call'}
PROPERTY ClassName : REFERENCE TO STRING
GET
ClassName REF= _ClassName;
END_GET
END_PROPERTY

METHOD FB_init : BOOL
VAR_INPUT
	bInitRetains : BOOL; // TRUE: the retain variables are initialized (reset warm / reset cold)
	bInCopyCode : BOOL;  // TRUE: the instance will be copied to the copy code afterward (online change)
	name : WSTRING;
END_VAR
END_METHOD

{attribute 'monitoring' := 'call'}
PROPERTY NamespaceName : REFERENCE TO STRING
GET
NamespaceName REF= CurrentNamespace.Name;
END_GET
END_PROPERTY

{attribute 'monitoring' := 'call'}
PROPERTY SelfSize : ULINT
GET
SelfSize := XSIZEOF(THIS^);
END_GET
END_PROPERTY

END_FUNCTION_BLOCK

// ---- Tests/JSON/JsonConfigurationTestRunner.TcPOU
(*
SPDX-FileCopyrightText: © 2026 Oleksandr Tiutyk <trofimich@gmail.com>
SPDX-License-Identifier: MIT
License: https://opensource.org/license/mit
*)

(*!
<summary>Runs the OpenFramework test groups registered by the shared test controller.</summary>
<description>
Owns persistent root instances and fixed child storage. The IO model group borrows the controller-owned fixture.
Use from one task without reentry.
Children borrows the same array for the instance lifetime. Root parents remain zero.
</description>
*)

{attribute 'no_assign'}
{attribute 'no_explicit_call' := 'do not call this function block directly'}
FUNCTION_BLOCK JsonConfigurationTestRunner EXTENDS TOF_Testing.TestRunner<45>
VAR_STAT
	//! <summary>Class name shared by instances of this concrete runner.</summary>
	{attribute 'hide'}
	_ClassName : STRING := __POUNAME();
END_VAR
VAR
	{attribute 'hide'}
	{attribute 'init_namespace'}
	_NamespaceName : STRING;
	//! <summary>Stable interface storage borrowed by the IO model group.</summary>
	_IOModelsFixture : IIOModelsTestFixture;
END_VAR
VAR_OUTPUT
	//! <summary>Owned root test suite for writer operations.</summary>
	WriterTest : JsonConfigurationWriterTest(name := "JsonConfigurationWriterTest", parent := 0);
	//! <summary>Owned root test suite for reader operations.</summary>
	ReaderTest : JsonConfigurationReaderTest(name := "JsonConfigurationReaderTest", parent := 0);
	//! <summary>Owned root test suite for round-trip serialization.</summary>
	RoundTripTest : JsonConfigurationRoundTripTest(name := "JsonConfigurationRoundTripTest", parent := 0);
	//! <summary>Owned root group for analog range conversions.</summary>
	RangeConverterTest : RangeAnalogValueConverterTest(name := "RangeAnalogValueConverterTest", parent := 0);
	//! <summary>Checks the two-cycle restart of an active timer.</summary>
	TimerRestartTest : TimerRestartWhileRunningTest(name := "RestartWhileRunning", parent := 0);
	//! <summary>Exercises failure to open a missing file for reading in an owned directory.</summary>
	MissingFileTest : OpenMissingFileForReadingTest(name := "OpenMissingFileForReading", parent := 0);
	//! <summary>Checks lexical file and directory path rules without filesystem I/O.</summary>
	PathValidationTest : LexicalPathValidationTest(name := "LexicalPathValidation", parent := 0);
	//! <summary>Groups the six filesystem contract tests that exercise no native I/O.</summary>
	FileSystemTests : FileSystemContractTest(name := "FileSystemContractTest", parent := 0);
	//! <summary>Groups the three native directory lifecycle scenarios.</summary>
	DirectoryTests : DirectoryTest(name := "DirectoryTest", parent := 0);
	//! <summary>Groups the four cyclic file-content manager scenarios.</summary>
	FileContentTests : FileContentManagerOperationsTest(name := "FileContentManagerTest", parent := 0);
	//! <summary>Groups the three native filesystem integration scenarios.</summary>
	FileSystemIntegrationTests : FileSystemIntegrationTestGroup(name := "FileSystemIntegrationTest", parent := 0);
	//! <summary>Groups the deterministic logger contracts and task-routing tests.</summary>
	LoggerContractTests : LoggerContractTestGroup(name := "LoggerContractTest", parent := 0);
	//! <summary>Runs the native file and EventLogger integration cases.</summary>
	LoggerIntegrationTests : LoggerIntegrationTestGroup(name := "LoggerTest", parent := 0);
	//! <summary>Groups the task lifecycle view and naming cases.</summary>
	TaskLifecycleTests : TaskLifecycleViewsTestGroup(name := "TaskLifecycleViewsTest", parent := 0);
	//! <summary>Groups FIFO and empty-queue behavior.</summary>
	TaskSequenceTests : TaskSequenceTestGroup(name := "TaskSequenceTest", parent := 0);
	//! <summary>Groups cooperative queue cleanup and failure cases.</summary>
	TaskQueueCleanupTests : TaskQueueCleanupTestGroup(name := "TaskQueueCleanupTest", parent := 0);
	//! <summary>Groups timer timing, lifecycle and restart cases.</summary>
	TimerTimingTests : TimerTimingTestGroup(name := "TimerTimingTest", parent := 0);
	//! <summary>Groups task stopping, failure and naming cases.</summary>
	TaskStoppingTests : TaskStoppingTestGroup(name := "TaskStoppingTest", parent := 0);
	//! <summary>Groups concrete object disposal and address conversion cases.</summary>
	ObjectLifetimeTests : ObjectLifetimeTestGroup(name := "ObjectLifetimeTest", parent := 0);
	//! <summary>Groups generic storage, ordering, conversion and runtime type diagnostics.</summary>
	GenericValueTests : GenericValueTestGroup(name := "GenericValueTest", parent := 0);
	//! <summary>Groups random range and dispersion contracts.</summary>
	RandomTests : RandomTestGroup(name := "RandomTest", parent := 0);
	//! <summary>Groups exception transport, cloning, diagnostics and failure boundaries.</summary>
	ExceptionTests : ExceptionTestGroup(name := "ExceptionTest", parent := 0);
	//! <summary>Groups byte-string formatting, editing, search and splitter contracts.</summary>
	StringTests : StringsTestGroup(name := "StringsTest", parent := 0);
	//! <summary>Groups wide-string formatting, editing, search and splitter contracts.</summary>
	WideStringTests : WideStringsTestGroup(name := "WideStringsTest", parent := 0);
	//! <summary>Groups byte-string builder assignment, reuse and failure contracts.</summary>
	StringBuilderTests : StringBuilderTestGroup(name := "StringBuilderTest", parent := 0);
	//! <summary>Groups wide-string builder assignment, reuse and failure cases.</summary>
	WideStringBuilderTests : WideStringBuilderTestGroup(name := "WideStringBuilderTest", parent := 0);
	//! <summary>Groups byte-list operations with dynamically allocated storage.</summary>
	DynamicByteListTests : DynamicByteListTestGroup(name := "DynamicByteListTest", parent := 0);
	//! <summary>Groups fixed-capacity byte-list operations and overflow handling.</summary>
	StaticByteListTests : StaticByteListTestGroup(name := "StaticByteListTest", parent := 0);
	//! <summary>Groups native JSON conversion, capacity, encoding and callback cases.</summary>
	AutomaticJsonSerializerTests : AutomaticJsonSerializerTestGroup(name := "AutomaticJsonSerializerTest", parent := 0);
	//! <summary>Groups fixed-capacity queue lookup, FIFO, clear and overflow cases.</summary>
	StaticQueueTests : StaticQueueTestGroup(name := "StaticQueueTest", parent := 0);
	//! <summary>Groups dynamic queue lookup, FIFO, growth and clear cases.</summary>
	DynamicQueueTests : DynamicQueueTestGroup(name := "DynamicQueueTest", parent := 0);
	//! <summary>Groups dynamic dictionary lookup, update, removal and clear cases.</summary>
	DynamicDictionaryTests : DynamicDictionaryTestGroup(name := "DynamicDictionaryTest", parent := 0);
	//! <summary>Groups fixed-capacity dictionary lookup, update, removal, clear and overflow cases.</summary>
	StaticDictionaryTests : StaticDictionaryTestGroup(name := "StaticDictionaryTest", parent := 0);
	//! <summary>Groups dynamic set lookup, duplicate updates, removal and clear cases.</summary>
	DynamicUniqueDataSetTests : DynamicUniqueDataSetTestGroup(name := "DynamicUniqueDataSetTest", parent := 0);
	//! <summary>Groups fixed-capacity set lookup, duplicate updates, removal, clear and overflow cases.</summary>
	StaticUniqueDataSetTests : StaticUniqueDataSetTestGroup(name := "StaticUniqueDataSetTest", parent := 0);
	//! <summary>Groups dynamic list copying, borrowing, editing, search, sorting and clear cases.</summary>
	DynamicListTests : DynamicListTestGroup(name := "DynamicListTest", parent := 0);
	//! <summary>Groups fixed-capacity list copying, borrowing, editing, search, sorting and overflow cases.</summary>
	StaticListTests : StaticListTestGroup(name := "StaticListTest", parent := 0);
	//! <summary>Groups dynamic stack storage, LIFO order, cursors and ownership cases.</summary>
	DynamicStackTests : DynamicStackTestGroup(name := "DynamicStackTest", parent := 0);
	//! <summary>Groups fixed-capacity stack storage, LIFO order, cursors, ownership and overflow cases.</summary>
	StaticStackTests : StaticStackTestGroup(name := "StaticStackTest", parent := 0);
	//! <summary>Groups digital and analog device, simulated channel and conversion cases.</summary>
	DevicesIOTests : DevicesIOTestGroup(name := "DevicesIOTest", parent := 0);
	//! <summary>Groups collection ownership, callback, growth and enumeration scenarios.</summary>
	CollectionsContractTests : CollectionsContractTestGroup(name := "CollectionsContractTest", parent := 0);
	//! <summary>Groups PDO representation and simulated input binding scenarios.</summary>
	IOModelsTests : IOModelsTestGroup(name := "IOModelsTest", parent := 0, fixtureSlot := ADR(_IOModelsFixture));
	//! <summary>Groups workflow integration, comparison and variable-scope scenarios.</summary>
	WorkflowComprehensiveTests : WorkflowComprehensiveTestGroup(name := "WorkflowComprehensiveTest", parent := 0);
	//! <summary>Groups workflow contracts and the cyclic delay timing regression.</summary>
	WorkflowContractTests : WorkflowContractTestGroup(name := "WorkflowContractTest", parent := 0);
	//! <summary>Groups automation component contracts and observations from the dedicated runner task.</summary>
	AutomationComponentTests : AutomationComponentTestGroup(name := "AutomationComponentTest", parent := 0);
END_VAR
VAR
	_Children : ARRAY [0.._ChildCount - 1] OF TOF_Testing.ITestElement :=
	[
		WriterTest,
		ReaderTest,
		RoundTripTest,
		RangeConverterTest,
		TimerRestartTest,
		MissingFileTest,
		PathValidationTest,
		FileSystemTests,
		DirectoryTests,
		FileContentTests,
		FileSystemIntegrationTests,
		LoggerContractTests,
		LoggerIntegrationTests,
		TaskLifecycleTests,
		TaskSequenceTests,
		TaskQueueCleanupTests,
		TimerTimingTests,
		TaskStoppingTests,
		ObjectLifetimeTests,
		GenericValueTests,
		RandomTests,
		ExceptionTests,
		StringTests,
		WideStringTests,
		StringBuilderTests,
		WideStringBuilderTests,
		DynamicByteListTests,
		StaticByteListTests,
		AutomaticJsonSerializerTests,
		StaticQueueTests,
		DynamicQueueTests,
		DynamicDictionaryTests,
		StaticDictionaryTests,
		DynamicUniqueDataSetTests,
		StaticUniqueDataSetTests,
		DynamicListTests,
		StaticListTests,
		DynamicStackTests,
		StaticStackTests,
		DevicesIOTests,
		CollectionsContractTests,
		IOModelsTests,
		WorkflowComprehensiveTests,
		WorkflowContractTests,
		AutomationComponentTests
	];
END_VAR

(*!
<summary>Stores the controller-owned model fixture for the IO model group.</summary>
<description>Stores a borrow without invoking the fixture. The controller keeps it alive for all test runs.</description>
<param name="ioModelsFixture">Controller-owned model fixture declared before the runner.</param>
*)
METHOD FB_init : BOOL
VAR_INPUT
	bInitRetains: BOOL; // TRUE: the retain variables are initialized (reset warm / reset cold)
	bInCopyCode: BOOL; // TRUE: the instance will be copied to the copy code afterward (online change)
	ioModelsFixture : IIOModelsTestFixture;
END_VAR
IF NOT bInCopyCode THEN
	_IOModelsFixture := ioModelsFixture;
END_IF

FB_init := TRUE;
END_METHOD

(*!
<summary>Borrows the unchanged persistent root array; application code must not modify it.</summary>
*)
{attribute 'monitoring' := 'call'}
PROPERTY Children : REFERENCE TO ARRAY [0.._ChildCount - 1] OF TOF_Testing.ITestElement
GET
Children REF= _Children;
END_GET
END_PROPERTY

(*!
<summary>Borrows the concrete class name; callers must not modify the returned storage.</summary>
*)
{attribute 'monitoring' := 'call'}
PROPERTY ClassName : REFERENCE TO STRING
GET
ClassName REF= _ClassName;
END_GET
END_PROPERTY

(*!
<summary>Borrows the concrete namespace name for the instance lifetime; callers must not modify it.</summary>
*)
{attribute 'monitoring' := 'call'}
PROPERTY NamespaceName : REFERENCE TO STRING
GET
NamespaceName REF= _NamespaceName;
END_GET
END_PROPERTY

(*!
<summary>Reports the complete concrete instance size in bytes.</summary>
*)
{attribute 'monitoring' := 'call'}
PROPERTY SelfSize : ULINT
GET
SelfSize := XSIZEOF(THIS^);
END_GET
END_PROPERTY

END_FUNCTION_BLOCK

// ---- Tests/JSON/JsonConfigurationWriterTest.TcPOU
(*
SPDX-FileCopyrightText: © 2026 Oleksandr Tiutyk <trofimich@gmail.com>
SPDX-License-Identifier: MIT
License: https://opensource.org/license/mit
*)

(*!
<summary>Exercises JsonConfigurationWriter serialization contracts, structural calls and failure handling.</summary>
<description>
Tests serialize invocation, exception recovery and reuse, null source rejection, argument validation,
manual document streaming, and destination buffer overflow detection.
</description>
*)

{attribute 'no_assign'}
{attribute 'no_explicit_call' := 'do not call this function block directly'}
FUNCTION_BLOCK JsonConfigurationWriterTest EXTENDS TOF_Testing.SingleCycleTest
VAR CONSTANT
	//! <summary>E_INVALIDARG identifies a rejected writer operand.</summary>
	_InvalidArgument : UDINT := 16#80070057;
END_VAR
VAR_STAT
	{attribute 'hide'}
	_ClassName : STRING := __POUNAME();
END_VAR
VAR
	{attribute 'hide'}
	{attribute 'init_namespace'}
	_NamespaceName : STRING;
END_VAR
VAR
	_Writer : TOF_JSON.JsonConfigurationWriter;
	_Dom : Tc3_JsonXml.FB_JsonDomParser;
	_Mock : MockConfigurationWritable;
	_Doc : TOF_Core.JSON_DOCUMENT;
END_VAR

(*!
<summary>Checks the source message of a caught framework exception and its HRESULT when specified.</summary>
<description>Reads the payload in the current task before cleanup. A missing or unrelated payload fails the test.</description>
*)
METHOD PRIVATE checkCaughtException
VAR_INPUT
	exceptionCode : __SYSTEM.ExceptionCode;
	expectedMessage : WSTRING(255);
	scenario : WSTRING(255);
	expectedCode : UDINT := 0;
END_VAR
VAR
	exception : TOF_Core.IException;
	generalException : TOF_Core.IGeneralException;
	diagnostic : TOF_Core.ERROR_MESSAGE;
END_VAR
exception := TOF_Core.ExceptionManager.GetLastException(
	exceptionCode := exceptionCode,
	catchPointNamespaceName := NamespaceName,
	catchPointPOUName := __POUNAME(),
	catchPointPosition := __POSITION()
);

IF exception = 0 OR_ELSE NOT __QUERYINTERFACE(exception, generalException) THEN
	diagnostic := TOF_Core.WideStrings.Concat255(scenario, ": expected a framework exception");
	RecordFailure(message := diagnostic);

	RETURN;
END_IF

Assert.ThatWideString(actual := generalException.SourceMessage, message := scenario).ToBe(expected := expectedMessage);

IF expectedCode <> TOF_Core.UnsignedInt32.ZERO THEN
	Assert.ThatUDInt(actual := generalException.ErrorCode, message := scenario).ToBe(expected := expectedCode);
END_IF
END_METHOD

(*!
<summary>Borrows the concrete class name for the lifetime of this instance.</summary>
*)
{attribute 'monitoring' := 'call'}
PROPERTY ClassName : REFERENCE TO STRING
GET
ClassName REF= _ClassName;
END_GET
END_PROPERTY

(*!
<summary>Exercises serialization, operand rejection and writer recovery in a single PLC cycle.</summary>
*)
METHOD PROTECTED ExecuteTest
testSerializeWritable();
testSerializeFailureClearsDocumentAndAllowsReuse();
testSerializeNullSource();
testInvalidValueOperands();
testDocumentBufferOverflow();
testManualDocumentConstruction();
END_METHOD

(*!
<summary>Requires the invalid-argument HRESULT when writing a DINT with the supplied source and size.</summary>
*)
METHOD PRIVATE expectInvalidValueOperand
VAR_INPUT
	name : STRING;
	data : PVOID;
	size : UDINT;
END_VAR
VAR
	exceptionCode : __SYSTEM.ExceptionCode;
	diagnostic : TOF_Core.ERROR_MESSAGE;
END_VAR
__TRY
	_Writer.WriteValue(
		name := name,
		valueType := TOF_Core.CONFIGURATION_VALUE_TYPE.TYPE_DINT,
		data := data,
		size := size
	);

	diagnostic := TOF_Core.WideStrings.Concat255("Writer accepted invalid operand: ", TO_WSTRING(name));
	RecordFailure(message := diagnostic);
__CATCH(exceptionCode)
	checkCaughtException(
		exceptionCode := exceptionCode,
		expectedMessage := "Cannot write configuration document",
		expectedCode := _InvalidArgument,
		scenario := TO_WSTRING(name)
	);
__ENDTRY
END_METHOD

(*!
<summary>Borrows the compiler-initialized namespace for the lifetime of this instance.</summary>
*)
{attribute 'monitoring' := 'call'}
PROPERTY NamespaceName : REFERENCE TO STRING
GET
NamespaceName REF= CurrentNamespace.Name;
END_GET
END_PROPERTY

(*!
<summary>Reports the complete concrete instance size in bytes.</summary>
*)
{attribute 'monitoring' := 'call'}
PROPERTY SelfSize : ULINT
GET
SelfSize := XSIZEOF(THIS^);
END_GET
END_PROPERTY

(*!
<summary>Checks the writer diagnostic when the serialized document exceeds the destination capacity.</summary>
<description>The array's string contents alone exceed the byte size of the destination buffer.</description>
*)
METHOD PRIVATE testDocumentBufferOverflow
VAR
	i : UDINT;
	itemCount : UDINT;
	value : STRING(50) := '01234567890123456789012345678901234567890123456789';
	exceptionCode : __SYSTEM.ExceptionCode;
END_VAR
_Writer.BeginDocument();
_Writer.BeginArray(name := 'overflowList');

itemCount := SIZEOF(_Doc) / TOF_Core.Strings.GetLength(value := value) + 1;

// SA0175: Raw string buffer passed to test document overflow; no character indexing.
{analysis -175}
FOR i := 1 TO itemCount DO
	_Writer.WriteValue(
		name := '',
		valueType := TOF_Core.CONFIGURATION_VALUE_TYPE.TYPE_STRING,
		data := ADR(value),
		size := SIZEOF(value)
	);
END_FOR
{analysis +175}

_Writer.EndArray();

__TRY
	_Writer.EndDocument(document := _Doc);
	RecordFailure(message := "Expected failure: Oversized document");
__CATCH(exceptionCode)
	checkCaughtException(
		exceptionCode := exceptionCode,
		expectedMessage := "Cannot write configuration document",
		scenario := "Oversized document"
	);
__ENDTRY
END_METHOD

(*!
<summary>Checks that rejected inputs leave a valid object ready for its next field.</summary>
*)
METHOD PRIVATE testInvalidValueOperands
VAR
	value : DINT := 123;
	root : Tc3_JsonXml.SJsonValue;
	member : Tc3_JsonXml.SJsonValue;
END_VAR
_Writer.BeginDocument();
expectInvalidValueOperand(name := 'nullData', data := 0, size := SIZEOF(value));
expectInvalidValueOperand(name := 'zeroSize', data := ADR(value), size := 0);
expectInvalidValueOperand(name := 'invalidSize', data := ADR(value), size := 3);
_Writer.WriteValue(
	name := 'valid',
	valueType := TOF_Core.CONFIGURATION_VALUE_TYPE.TYPE_DINT,
	data := ADR(value),
	size := SIZEOF(value)
);
_Writer.EndDocument(document := _Doc);

root := _Dom.ParseDocument(sJson := _Doc);

IF root = 0 OR_ELSE NOT _Dom.IsObject(v := root) THEN
	RecordFailure(message := "Rejected fields must leave the writer able to finish a valid object");
	RETURN;
END_IF

IF _Dom.FindMember(v := root, member := 'nullData') <> 0
	OR_ELSE _Dom.FindMember(v := root, member := 'zeroSize') <> 0
	OR_ELSE _Dom.FindMember(v := root, member := 'invalidSize') <> 0
THEN
	RecordFailure(message := "A rejected argument emitted a property key");
	RETURN;
END_IF

member := _Dom.FindMember(v := root, member := 'valid');

IF member = 0 OR_ELSE NOT _Dom.IsInt(v := member) THEN
	RecordFailure(message := "Expected the next valid field to contain an integer");
	RETURN;
END_IF

Assert.ThatDInt(actual := _Dom.GetInt(v := member), message := "Value after rejected operands").ToBe(expected := value);
END_METHOD

(*!
<summary>Verifies the shape and values produced by manual object and array streaming.</summary>
*)
METHOD PRIVATE testManualDocumentConstruction
VAR
	val : DINT := 10;
	item : DINT := 1;
	root : Tc3_JsonXml.SJsonValue;
	cfg : Tc3_JsonXml.SJsonValue;
	items : Tc3_JsonXml.SJsonValue;
	value : Tc3_JsonXml.SJsonValue;
END_VAR
_Writer.BeginDocument();

_Writer.BeginObject(name := 'cfg');
_Writer.WriteValue(
	name := 'num',
	valueType := TOF_Core.CONFIGURATION_VALUE_TYPE.TYPE_DINT,
	data := ADR(val),
	size := SIZEOF(val)
);
_Writer.EndObject();

_Writer.BeginArray(name := 'items');
_Writer.WriteValue(
	name := '',
	valueType := TOF_Core.CONFIGURATION_VALUE_TYPE.TYPE_DINT,
	data := ADR(item),
	size := SIZEOF(item)
);
_Writer.EndArray();

_Writer.EndDocument(document := _Doc);

root := _Dom.ParseDocument(sJson := _Doc);
IF root = 0 OR_ELSE NOT _Dom.IsObject(v := root) THEN
	RecordFailure(message := "Manual serialization must produce a JSON object");
	RETURN;
END_IF

cfg := _Dom.FindMember(v := root, member := 'cfg');

IF cfg = 0 OR_ELSE NOT _Dom.IsObject(v := cfg) THEN
	RecordFailure(message := "cfg must be a nested JSON object");
	RETURN;
END_IF

value := _Dom.FindMember(v := cfg, member := 'num');

IF value = 0 OR_ELSE NOT _Dom.IsInt(v := value) THEN
	RecordFailure(message := "cfg.num must be a JSON integer");
	RETURN;
END_IF

Assert.ThatDInt(actual := _Dom.GetInt(v := value), message := "cfg.num value").ToBe(expected := 10);

items := _Dom.FindMember(v := root, member := 'items');
IF items = 0 OR_ELSE NOT _Dom.IsArray(v := items) THEN
	RecordFailure(message := "items must be a JSON array");
	RETURN;
END_IF

IF _Dom.GetArraySize(v := items) <> 1 THEN
	RecordFailure(message := "items must contain exactly one element");
	RETURN;
END_IF

value := _Dom.GetArrayValueByIdx(v := items, idx := 0);
IF value = 0 OR_ELSE NOT _Dom.IsInt(v := value) THEN
	RecordFailure(message := "items[0] must be a JSON integer");
	RETURN;
END_IF

Assert.ThatDInt(actual := _Dom.GetInt(v := value), message := "items[0] value").ToBe(expected := 1);
END_METHOD

(*!
<summary>Checks propagation of the callback failure, document clearing, and reuse without manual reset.</summary>
*)
METHOD PRIVATE testSerializeFailureClearsDocumentAndAllowsReuse
VAR
	exceptionCode : __SYSTEM.ExceptionCode;
	hasContent : BOOL;
END_VAR
_Mock.Reset();
_Mock.ThrowOnSerialize := TRUE;
_Doc := 'pre-existing content that must be cleared';

__TRY
	_Writer.Serialize(source := _Mock, document := _Doc);
	RecordFailure(message := "Expected failure: Throwing serialization callback");
__CATCH(exceptionCode)
	checkCaughtException(
		exceptionCode := exceptionCode,
		expectedMessage := "Mock serialize failure",
		scenario := "Throwing serialization callback"
	);
__ENDTRY

Assert.ThatString(actual := _Doc).ToBe(expected := '');

_Mock.ThrowOnSerialize := FALSE;
_Writer.Serialize(source := _Mock, document := _Doc);

hasContent := Tc2_Standard.LEN(STR := _Doc) > 0;
Assert.ThatBool(actual := hasContent).IsTrue();
Assert.ThatUDInt(actual := _Mock.SerializeCount).ToBe(expected := 1);
END_METHOD

(*!
<summary>Requires the invalid-argument diagnostic for a null serialization source.</summary>
*)
METHOD PRIVATE testSerializeNullSource
VAR
	nullSource : TOF_Core.IConfigurationSerializable := 0;
	exceptionCode : __SYSTEM.ExceptionCode;
END_VAR
__TRY
	_Writer.Serialize(source := nullSource, document := _Doc);
	RecordFailure(message := "Expected failure: Null serialization source");
__CATCH(exceptionCode)
	checkCaughtException(
		exceptionCode := exceptionCode,
		expectedMessage := "Cannot write configuration document",
		expectedCode := _InvalidArgument,
		scenario := "Null serialization source"
	);
__ENDTRY
END_METHOD

(*!
<summary>Verifies the serialized object values and JSON types with the native DOM parser.</summary>
*)
METHOD PRIVATE testSerializeWritable
VAR
	root : Tc3_JsonXml.SJsonValue;
	value : Tc3_JsonXml.SJsonValue;
END_VAR
_Mock.Reset();
_Writer.Serialize(source := _Mock, document := _Doc);
Assert.ThatUDInt(actual := _Mock.SerializeCount).ToBe(expected := 1);

root := _Dom.ParseDocument(sJson := _Doc);
IF root = 0 OR_ELSE NOT _Dom.IsObject(v := root) THEN
	RecordFailure(message := "Object serialization must produce a JSON object");
	RETURN;
END_IF

value := _Dom.FindMember(v := root, member := 'intField');
IF value = 0 OR_ELSE NOT _Dom.IsInt(v := value) THEN
	RecordFailure(message := "intField must be a JSON integer");
	RETURN;
END_IF

Assert.ThatDInt(actual := _Dom.GetInt(v := value), message := "intField value").ToBe(expected := 42);

value := _Dom.FindMember(v := root, member := 'stringField');
IF value = 0 OR_ELSE NOT _Dom.IsString(v := value) THEN
	RecordFailure(message := "stringField must be a JSON string");
	RETURN;
END_IF

Assert.ThatString(actual := _Dom.GetString(v := value), message := "stringField value").ToBe(expected := 'hello');
END_METHOD

END_FUNCTION_BLOCK

// ---- Tests/JSON/MockConfigurationWritable.TcPOU
(*
SPDX-FileCopyrightText: © 2026 Oleksandr Tiutyk <trofimich@gmail.com>
SPDX-License-Identifier: MIT
License: https://opensource.org/license/mit
*)

(*!
<summary>Mock configuration serializable object for writer and round-trip tests.</summary>
<description>
Provides controlled serialization and deserialization with optional failure injection.
Used exclusively by JSON configuration unit tests.
</description>
*)

{attribute 'no_explicit_call' := 'do not call this function block directly'}
FUNCTION_BLOCK MockConfigurationWritable EXTENDS TOF_Core.Object IMPLEMENTS TOF_Core.IConfigurationSerializable
VAR_STAT
	{attribute 'hide'}
	_ClassName : STRING := __POUNAME();
END_VAR
VAR
	{attribute 'hide'}
	{attribute 'init_namespace'}
	_NamespaceName : STRING;
END_VAR
VAR_INPUT
	ThrowOnSerialize : BOOL;
	IntField : DINT := 42;
	StringField : STRING(80) := 'hello';
	WriteNestedObject : BOOL;
	WriteArray : BOOL;
END_VAR
VAR_OUTPUT
	SerializeCount : UDINT;
	DeserializeCount : UDINT;
END_VAR

(*!
<summary>Borrows the concrete class name for the lifetime of this instance.</summary>
*)
{attribute 'monitoring' := 'call'}
PROPERTY ClassName : REFERENCE TO STRING
GET
ClassName REF= _ClassName;
END_GET
END_PROPERTY

(*!
<summary>Restores fields from the configuration reader.</summary>
<description>
The reader and document node are borrowed for this call. The deserialization context is ignored.
</description>
<param name="reader">Active configuration reader.</param>
<param name="node">Object node to read fields from.</param>
<param name="context">Configuration deserialization context; ignored by this mock.</param>
*)
METHOD Deserialize
VAR_INPUT
	reader : TOF_Core.IConfigurationReader;
	node : TOF_Core.CONFIGURATION_NODE;
	context : TOF_Core.IConfigurationDeserializationContext;
END_VAR
VAR
	fieldNode : TOF_Core.CONFIGURATION_NODE;
END_VAR
DeserializeCount := DeserializeCount + 1;
fieldNode := reader.GetField(node := node, name := 'intField');
reader.ReadValue(
	node := fieldNode,
	valueType := TOF_Core.CONFIGURATION_VALUE_TYPE.TYPE_DINT,
	data := ADR(IntField),
	size := SIZEOF(IntField)
);

fieldNode := reader.GetField(node := node, name := 'stringField');
// SA0175: Raw string buffer passed to ReadValue; no character indexing.
{analysis -175}
reader.ReadValue(
	node := fieldNode,
	valueType := TOF_Core.CONFIGURATION_VALUE_TYPE.TYPE_STRING,
	data := ADR(StringField),
	size := SIZEOF(StringField)
);
{analysis +175}
END_METHOD

(*!
<summary>Borrows the compiler-initialized namespace for the lifetime of this instance.</summary>
*)
{attribute 'monitoring' := 'call'}
PROPERTY NamespaceName : REFERENCE TO STRING
GET
NamespaceName REF= CurrentNamespace.Name;
END_GET
END_PROPERTY

(*!
<summary>Resets the mock state to defaults.</summary>
*)
METHOD Reset
ThrowOnSerialize := FALSE;
IntField := 42;
StringField := 'hello';
WriteNestedObject := FALSE;
WriteArray := FALSE;
SerializeCount := 0;
DeserializeCount := 0;
END_METHOD

(*!
<summary>Reports the complete concrete instance size in bytes.</summary>
*)
{attribute 'monitoring' := 'call'}
PROPERTY SelfSize : ULINT
GET
SelfSize := XSIZEOF(THIS^);
END_GET
END_PROPERTY

(*!
<summary>Writes mock state using the provided configuration writer.</summary>
<param name="writer">Target configuration writer.</param>
*)
METHOD Serialize
VAR_INPUT
	writer : TOF_Core.IConfigurationWriter;
END_VAR
VAR
	nestedValue : DINT := 999;
	arrayItem : DINT := 100;
END_VAR
IF ThrowOnSerialize THEN
	TOF_Core.Exceptions.ThrowStandard(
		sourceNamespaceName := NamespaceName,
		sourceClassName := ClassName,
		sourcePOUName := __POUNAME(),
		sourcePosition := __POSITION(),
		message := "Mock serialize failure"
	);
END_IF

SerializeCount := SerializeCount + 1;

writer.WriteValue(
	name := 'intField',
	valueType := TOF_Core.CONFIGURATION_VALUE_TYPE.TYPE_DINT,
	data := ADR(IntField),
	size := SIZEOF(IntField)
);

// SA0175: Raw string buffer passed to WriteValue; no character indexing.
{analysis -175}
writer.WriteValue(
	name := 'stringField',
	valueType := TOF_Core.CONFIGURATION_VALUE_TYPE.TYPE_STRING,
	data := ADR(StringField),
	size := SIZEOF(StringField)
);
{analysis +175}

IF WriteNestedObject THEN
	writer.BeginObject(name := 'nested');
	writer.WriteValue(
		name := 'nestedValue',
		valueType := TOF_Core.CONFIGURATION_VALUE_TYPE.TYPE_DINT,
		data := ADR(nestedValue),
		size := SIZEOF(nestedValue)
	);
	writer.EndObject();
END_IF

IF WriteArray THEN
	writer.BeginArray(name := 'arr');
	writer.WriteValue(
		name := '',
		valueType := TOF_Core.CONFIGURATION_VALUE_TYPE.TYPE_DINT,
		data := ADR(arrayItem),
		size := SIZEOF(arrayItem)
	);
	writer.EndArray();
END_IF
END_METHOD

END_FUNCTION_BLOCK

// ---- Tests/JSON/JsonConfigurationReaderTest.TcPOU
(*
SPDX-FileCopyrightText: © 2026 Oleksandr Tiutyk <trofimich@gmail.com>
SPDX-License-Identifier: MIT
License: https://opensource.org/license/mit
*)

(*!
<summary>Exercises JsonConfigurationReader document opening, member navigation and value reading error cases.</summary>
<description>
Verifies object root requirement, mandatory and optional field retrieval, list inspection, item bounds,
type and size mismatch detection, null rejection, buffer capacity checks, and repeated Open behavior.
</description>
*)

{attribute 'no_assign'}
{attribute 'no_explicit_call' := 'do not call this function block directly'}
FUNCTION_BLOCK JsonConfigurationReaderTest EXTENDS TOF_Testing.SingleCycleTest
VAR_STAT
	{attribute 'hide'}
	_ClassName : STRING := __POUNAME();
END_VAR
VAR
	{attribute 'hide'}
	{attribute 'init_namespace'}
	_NamespaceName : STRING;
END_VAR
VAR CONSTANT
	//! <summary>HRESULT for invalid arguments used by JsonConfigurationReader diagnostics.</summary>
	_InvalidArgumentCode : UDINT := 16#80070057;
END_VAR
VAR
	_Reader : TOF_JSON.JsonConfigurationReader;
	_Mock : MockConfigurationWritable;
	_Doc : TOF_Core.JSON_DOCUMENT;
END_VAR

(*!
<summary>Borrows the concrete class name for the lifetime of this instance.</summary>
*)
{attribute 'monitoring' := 'call'}
PROPERTY ClassName : REFERENCE TO STRING
GET
ClassName REF= _ClassName;
END_GET
END_PROPERTY

(*!
<summary>Executes reader scenarios including Unicode decoding and destination capacity in a single PLC cycle.</summary>
*)
METHOD PROTECTED ExecuteTest
testOpenObjectRoot();
testOpenNonObjectRoot();
testOpenInvalidJson();
testFieldExistingAndMissing();
testFieldOnNonObject();
testFindOptionalField();
testListOperations();
testReadValueValidationAndErrors();
testReadWideString();
testReparseReadsNewDocument();
testDeserializeContextFreeObject();
END_METHOD

(*!
<summary>Borrows the compiler-initialized namespace for the lifetime of this instance.</summary>
*)
{attribute 'monitoring' := 'call'}
PROPERTY NamespaceName : REFERENCE TO STRING
GET
NamespaceName REF= CurrentNamespace.Name;
END_GET
END_PROPERTY

(*!
<summary>Reports the complete concrete instance size in bytes.</summary>
*)
{attribute 'monitoring' := 'call'}
PROPERTY SelfSize : ULINT
GET
SelfSize := XSIZEOF(THIS^);
END_GET
END_PROPERTY

(*!
<summary>Verifies mandatory field lookup and missing field exception.</summary>
*)
METHOD PRIVATE testFieldExistingAndMissing
VAR
	root : TOF_Core.CONFIGURATION_NODE;
	fieldNode : TOF_Core.CONFIGURATION_NODE;
	caughtMessage : WSTRING(255);
	exceptionCode : __SYSTEM.ExceptionCode;
END_VAR
_Doc := '{"existing": 42}';
root := _Reader.Parse(document := _Doc);

fieldNode := _Reader.GetField(node := root, name := 'existing');
Assert.ThatBool(actual := _Reader.IsPresent(node := fieldNode)).IsTrue();

caughtMessage := TOF_Core.WideStrings.Empty;

__TRY
	fieldNode := _Reader.GetField(node := root, name := 'missing');
__CATCH(exceptionCode)
	caughtMessage := getInvalidDocumentMessage(
		exceptionCode := exceptionCode,
		catchPointPOUName := __POUNAME(),
		catchPointPosition := __POSITION()
	);
__ENDTRY

Assert.ThatWideString(
	actual := caughtMessage,
	message := "GetField on a missing member"
).ToBe(expected := "Invalid JSON configuration: missing field (field: missing)");
END_METHOD

(*!
<summary>Verifies that Field on a non-object parent raises not an object.</summary>
*)
METHOD PRIVATE testFieldOnNonObject
VAR
	root : TOF_Core.CONFIGURATION_NODE;
	scalarNode : TOF_Core.CONFIGURATION_NODE;
	childNode : TOF_Core.CONFIGURATION_NODE;
	caughtMessage : WSTRING(255);
	exceptionCode : __SYSTEM.ExceptionCode;
END_VAR
_Doc := '{"scalar": 42}';
root := _Reader.Parse(document := _Doc);
scalarNode := _Reader.GetField(node := root, name := 'scalar');

caughtMessage := TOF_Core.WideStrings.Empty;

__TRY
	childNode := _Reader.GetField(node := scalarNode, name := 'child');
__CATCH(exceptionCode)
	caughtMessage := getInvalidDocumentMessage(
		exceptionCode := exceptionCode,
		catchPointPOUName := __POUNAME(),
		catchPointPosition := __POSITION()
	);
__ENDTRY

Assert.ThatWideString(
	actual := caughtMessage,
	message := "GetField on a scalar"
).ToBe(expected := "Invalid JSON configuration: not an object (field: child)");
END_METHOD

(*!
<summary>Verifies IsList, Count, Item bounds and non-list error detection.</summary>
*)
METHOD PRIVATE testListOperations
VAR
	root : TOF_Core.CONFIGURATION_NODE;
	listNode : TOF_Core.CONFIGURATION_NODE;
	objNode : TOF_Core.CONFIGURATION_NODE;
	item0 : TOF_Core.CONFIGURATION_NODE;
	item2 : TOF_Core.CONFIGURATION_NODE;
	itemBad : TOF_Core.CONFIGURATION_NODE;
	countVal : UDINT;
	caughtMessage : WSTRING(255);
	exceptionCode : __SYSTEM.ExceptionCode;
END_VAR
_Doc := '{"list": [10, 20, 30], "obj": {"x": 1}}';
root := _Reader.Parse(document := _Doc);

listNode := _Reader.GetField(node := root, name := 'list');
Assert.ThatBool(actual := _Reader.IsArray(node := listNode)).IsTrue();
Assert.ThatUDInt(actual := _Reader.GetArraySize(node := listNode)).ToBe(expected := 3);

item0 := _Reader.GetItem(node := listNode, index := 0);
Assert.ThatBool(actual := _Reader.IsPresent(node := item0)).IsTrue();

item2 := _Reader.GetItem(node := listNode, index := 2);
Assert.ThatBool(actual := _Reader.IsPresent(node := item2)).IsTrue();

caughtMessage := TOF_Core.WideStrings.Empty;

__TRY
	itemBad := _Reader.GetItem(node := listNode, index := 3);
__CATCH(exceptionCode)
	caughtMessage := getInvalidDocumentMessage(
		exceptionCode := exceptionCode,
		catchPointPOUName := __POUNAME(),
		catchPointPosition := __POSITION()
	);
__ENDTRY

Assert.ThatWideString(
	actual := caughtMessage,
	message := "GetItem at the array length"
).ToBe(expected := "Invalid JSON configuration: index out of range");

objNode := _Reader.GetField(node := root, name := 'obj');
Assert.ThatBool(actual := _Reader.IsArray(node := objNode)).IsFalse();

caughtMessage := TOF_Core.WideStrings.Empty;

__TRY
	countVal := _Reader.GetArraySize(node := objNode);
__CATCH(exceptionCode)
	caughtMessage := getInvalidDocumentMessage(
		exceptionCode := exceptionCode,
		catchPointPOUName := __POUNAME(),
		catchPointPosition := __POSITION()
	);
__ENDTRY

Assert.ThatWideString(
	actual := caughtMessage,
	message := "GetArraySize on an object"
).ToBe(expected := "Invalid JSON configuration: not an array");

caughtMessage := TOF_Core.WideStrings.Empty;

__TRY
	itemBad := _Reader.GetItem(node := objNode, index := 0);
__CATCH(exceptionCode)
	caughtMessage := getInvalidDocumentMessage(
		exceptionCode := exceptionCode,
		catchPointPOUName := __POUNAME(),
		catchPointPosition := __POSITION()
	);
__ENDTRY

Assert.ThatWideString(
	actual := caughtMessage,
	message := "GetItem on an object"
).ToBe(expected := "Invalid JSON configuration: not an array");
END_METHOD

(*!
<summary>Verifies that Open raises parse failure on malformed JSON text.</summary>
*)
METHOD PRIVATE testOpenInvalidJson
VAR
	root : TOF_Core.CONFIGURATION_NODE;
	caughtMessage : WSTRING(255);
	exceptionCode : __SYSTEM.ExceptionCode;
END_VAR
_Doc := '{unclosed object';

caughtMessage := TOF_Core.WideStrings.Empty;

__TRY
	root := _Reader.Parse(document := _Doc);
__CATCH(exceptionCode)
	caughtMessage := getInvalidDocumentMessage(
		exceptionCode := exceptionCode,
		catchPointPOUName := __POUNAME(),
		catchPointPosition := __POSITION()
	);
__ENDTRY

Assert.ThatWideString(
	actual := caughtMessage,
	message := "Parse malformed JSON"
).ToBe(expected := "Invalid JSON configuration: parse failure");
END_METHOD

(*!
<summary>Verifies that Open rejects array or primitive roots.</summary>
*)
METHOD PRIVATE testOpenNonObjectRoot
VAR
	root : TOF_Core.CONFIGURATION_NODE;
	caughtMessage : WSTRING(255);
	exceptionCode : __SYSTEM.ExceptionCode;
END_VAR
_Doc := '[1, 2, 3]';

caughtMessage := TOF_Core.WideStrings.Empty;

__TRY
	root := _Reader.Parse(document := _Doc);
__CATCH(exceptionCode)
	caughtMessage := getInvalidDocumentMessage(
		exceptionCode := exceptionCode,
		catchPointPOUName := __POUNAME(),
		catchPointPosition := __POSITION()
	);
__ENDTRY

